(* Logix 5000 project; controller Comas_L4 vendor 1 type 14 code 193 rev 30.11; software revision 30.02 *)

TASK Gestion_Rapide (task) : Main
TASK MainTask (periodic, rate 5 ms, priority 10, watchdog 10 ms) : General, Comas

MODULES
   Local : vendor 1 type 14 code 193 (5069 0, rev 30.11)
      SortieF_4 : vendor 1 type 14 code 154 (Ethernet 172.10.3.20, rev 21.1)
      Var_Vertical_Droit : vendor 1 type 37 code 48 (Ethernet 172.10.12.22, rev 7.1, MotionDiagnostics RPI 1 ms, MotionSync RPI 5 ms)
      Var_Pompe_Doseuse : vendor 1 type 37 code 49 (Ethernet 172.10.12.20, rev 7.1, MotionSync RPI 5 ms, MotionDiagnostics RPI 1 ms)
      Var_Vertical_Gauche : vendor 1 type 37 code 48 (Ethernet 172.10.12.21, rev 7.1, MotionSync RPI 5 ms, MotionDiagnostics RPI 1 ms)
      Var_Rouleaux_Canneles : vendor 1 type 37 code 48 (Ethernet 172.10.12.26, rev 7.1, MotionDiagnostics RPI 1 ms, MotionSync RPI 5 ms)
      Codeur_Four : 842E-CM-M (Ethernet 172.10.12.19, rev 1.1, MotionDiagnostics RPI 1 ms, MotionSync RPI 5 ms)
      Var_Coupe_Fil : vendor 1 type 37 code 48 (Ethernet 172.10.12.25, rev 7.1, MotionSync RPI 5 ms, MotionDiagnostics RPI 1 ms)
      Var_Horizontal_Gauche : vendor 1 type 37 code 48 (Ethernet 172.10.12.23, rev 7.1, MotionSync RPI 5 ms, MotionDiagnostics RPI 1 ms)
      Var_Horizontal_Droit : vendor 1 type 37 code 48 (Ethernet 172.10.12.24, rev 7.1, MotionDiagnostics RPI 1 ms, MotionSync RPI 5 ms)
      Stratix_5700 : vendor 1 type 12 code 241 (Ethernet 172.10.12.13, rev 7.1, Output RPI 1000 ms)
      Entrees_2 : 5069-IB16 (5069 2, rev 2.1, StandardDataDriven RPI 5 ms)
      Entrees_1 : 5069-IB16 (5069 1, rev 2.1, StandardDataDriven RPI 5 ms)
      Sorties_1 : 5069-OB16 (5069 3, rev 2.1, StandardDataDriven RPI 5 ms)
END_MODULES

TYPE Chart :   // Chart Control Data Source
STRUCT
   Title : STRING;
   NumberOfDataPoints : INT;
   X_Axis_Label : STRING;
   X_Axis_Min : REAL;
   X_Axis_Max : REAL;
   Y_Axis_Label : STRING;
   Y_Axis_Min : REAL;
   Y_Axis_Max : REAL;
   DataSeries_FixedAxis : DataSeries;
   DataSeries_1 : DataSeries;
   DataSeries_2 : DataSeries;
   DataSeries_3 : DataSeries;
   DataSeries_4 : DataSeries;
   DataSeries_5 : DataSeries;
   DataSeries_6 : DataSeries;
   DataSeries_7 : DataSeries;
   DataSeries_8 : DataSeries;
END_STRUCT
END_TYPE

TYPE DataSeries :
STRUCT
   Label : STRING;
   Visible : BOOL;
   Data : REAL[500];
END_STRUCT
END_TYPE

TYPE UDT_Axis_Cam_Profil :
STRUCT
   Cam : CAM[80];
   MasterPeriode : REAL;
   SlavePeriode : REAL;
   NbrOfCamPoints : DINT;
   StartSlope : REAL;
   EndSlope : REAL;
   MasterScaling : REAL;
   SlaveScaling : REAL;
END_STRUCT
END_TYPE

TYPE UDT_CAM_PAN :
STRUCT
   A : UDT_CAM_POINT;
   B : UDT_CAM_POINT;
   C : UDT_CAM_POINT;
   D : UDT_CAM_POINT;
   E : UDT_CAM_POINT;
   F : UDT_CAM_POINT;
   G : UDT_CAM_POINT;
   H : UDT_CAM_POINT;
   I : UDT_CAM_POINT;
   J : UDT_CAM_POINT;
   K : UDT_CAM_POINT;
   L : UDT_CAM_POINT;
   M : UDT_CAM_POINT;
   N : UDT_CAM_POINT;
   O : UDT_CAM_POINT;
   P : UDT_CAM_POINT;
   Q : UDT_CAM_POINT;
   R : UDT_CAM_POINT;
   S : UDT_CAM_POINT;
   T : UDT_CAM_POINT;
   U : UDT_CAM_POINT;
   V : UDT_CAM_POINT;
   W : UDT_CAM_POINT;
   X : UDT_CAM_POINT;
   Y : UDT_CAM_POINT;
END_STRUCT
END_TYPE

TYPE UDT_CAM_POINT :
STRUCT
   x : REAL;
   y : REAL;
END_STRUCT
END_TYPE

TYPE UDT_CamGeneration :
STRUCT
   Cmd : UDT_CamGeneration_Cmd;
   In : UDT_CamGeneration_In;
   Out : UDT_CamGeneration_Out;
END_STRUCT
END_TYPE

TYPE UDT_CamGeneration_Cmd :
STRUCT
   Reset : BOOL;   // Effacement défaut
   Start : BOOL;   // Commande de lancement des calculs
   CamOrCamProfil : BOOL;   // 0 = tableau de points (sans MCCP) 1 = Profil executable (avec MCCP)
   Optimize : BOOL;
END_STRUCT
END_TYPE

TYPE UDT_CamGeneration_In :
STRUCT
   Cam : CAM[32];
   StartSlope : REAL;
   EndSlope : REAL;
   DefaultProfilType : INT;   // 2 = Modified Trapezoidal 4 = Sine modified 5 = 3-4-5 Poly 7 = 4-5-6-7 Poly
   Cfg_Segments : UDT_SegmentSetUp[32];
END_STRUCT
END_TYPE

TYPE UDT_CamGeneration_Out :
STRUCT
   Cam : CAM[32];
   NbrOfCamPoints : DINT;
   StartSlope : REAL;
   EndSlope : REAL;
   CamProfil : CAM_PROFILE[32];
END_STRUCT
END_TYPE

TYPE UDT_CamSegment :
STRUCT
   M0 : REAL;
   S0 : REAL;
   V0 : REAL;
   V1 : REAL;
   V2 : REAL;
   M1 : REAL;
   M2 : REAL;
   M3 : REAL;
   M4 : REAL;
   M5 : REAL;
   dM : REAL;
   a4 : REAL;
   S1 : REAL;
   S2 : REAL;
   S3 : REAL;
   S4 : REAL;
   S5 : REAL;
   dS : REAL;
   K1 : REAL;
   K2 : REAL;
   K3 : REAL;
   K4 : REAL;
   K5 : REAL;
   K6 : REAL;
   K7 : REAL;
   K8 : REAL;
   K9 : REAL;
   ActSlope : REAL;
   PrevSlope : REAL;
   No_Of_Points : DINT;
   NbPoints : DINT;
   CfgIndex : DINT;
   CAM_Points : CAM[32];
   Cv : REAL[2];
   Mn : REAL[2];
   Sn : REAL[2];
   RiseReturnComp : BOOL[32];
   IsAcceleration : BOOL;
   Err : BOOL;
   B1 : BOOL;
   MemoRiseReturnComp : BOOL;
END_STRUCT
END_TYPE

TYPE UDT_COM_Comas_Vers_SortieF :   // echange de donnée entre comas et sortie four
STRUCT
   Forage_Panel_O_F_Trappe : BOOL;
   ReserveBool : BOOL;
   ReserveBool2 : BOOL;
   ReserveReal : REAL;
   ReserveReal2 : REAL;
   ReserveReal3 : REAL;
END_STRUCT
END_TYPE

TYPE UDT_COMAS :
STRUCT
   Pas_Machine : DINT;
   Dephasage_Maitre : REAL;
   Came_Maitre : CAM[100];
   Longueur_Came_Maitre : DINT;
   Tete : UDT_COMAS_TETE;
   Pompe : UDT_COMAS_POMPE;
   Rouleaux : UDT_COMAS_ROULEAUX;
   Coupe_Fil : UDT_COMAS_COUPE;
   Start_Cam_Logique_Decoreuse : REAL;
   Stop_Cam_Logique_Decoreuse : REAL;
   Start_Cam_Logique_Doseuse : REAL;
   Stop_Cam_Logique_Doseuse : REAL;
   Consigne_Vitesse_Manu_mm : REAL;
   Consigne_Acc_Decc_Manu_mm : REAL;
   Consigne_Jerk_Manu : REAL;
   Activation_Cam_Auto : BOOL;
   Mode_CPT_Presence : BOOL;
   Distance_CPT_Presence_Produit : DINT;
   Consigne_Vitesse_Manu_Tour : REAL;
   Consigne_Acc_Decc_Manu_Tour : REAL;
   Distance_Decoreuse_mm : REAL;
   Distance_Doseuse_mm : REAL;
   Mode_Decoreuse_Cam_Logique : BOOL;
   Reserve_Real1 : REAL;
   Reserve_Real2 : REAL;
   Reserve_Real3 : REAL;
   Reserve_Real4 : REAL;
   Reserve_Real5 : REAL;
   Reserve_Bool1 : BOOL;
   Reserve_Bool2 : BOOL;
   Reserve_Bool3 : BOOL;
   Reserve_Bool4 : BOOL;
   Reserve_Bool5 : BOOL;
   Reserve_Real6 : REAL;
   Reserve_Real7 : REAL;
   Reserve_Real8 : REAL;
   Reserve_Real9 : REAL;
   Reserve_Real10 : REAL;
END_STRUCT
END_TYPE

TYPE UDT_COMAS_COUPE :
STRUCT
   Activation : BOOL;
   Start_Cam_Logique_Virtuelle : REAL;
   Stop_Cam_Logique_Virtuelle : REAL;
   Consigne_Vitesse_Virtuelle : REAL;
   Consigne_Acc_Dec_Virtuelle : REAL;
   Consigne_Jerk_Virtuelle : REAL;
   Cam_Axe : CAM[100];
   Longueur_Cam_Axe : DINT;
   Offset_Axe : REAL;
   Points_Pan : UDT_CAM_PAN;
   Reserve_Real1 : REAL;
   Reserve_Real2 : REAL;
   Reserve_Real3 : REAL;
   Reserve_Real4 : REAL;
   Reserve_Real5 : REAL;
   Reserve_Bool1 : BOOL;
   Reserve_Bool2 : BOOL;
   Reserve_Bool3 : BOOL;
   Reserve_Bool4 : BOOL;
   Reserve_Bool5 : BOOL;
END_STRUCT
END_TYPE

TYPE UDT_COMAS_POMPE :
STRUCT
   Start_Cam_Logique_Avance : REAL;
   Stop_Cam_Logique_Avance : REAL;
   Start_Cam_Logique_Recul : REAL;
   Stop_Cam_Logique_Recul : REAL;
   Consigne_Vitesse_Avance : REAL;
   Consigne_Acc_Dec_Avance : REAL;
   Consigne_Jerk_Avance : REAL;
   Consigne_Vitesse_Recul : REAL;
   Consigne_Acc_Dec_Recul : REAL;
   Consigne_Jerk_Recul : REAL;
   Offset_Axe : REAL;
   Points_Pan : UDT_CAM_PAN;
   Start_Cam_Logique_Inter1 : REAL;
   Stop_Cam_Logique_Inter1 : REAL;
   Consigne_Vitesse_Inter1 : REAL;
   Start_Cam_Logique_Inter2 : REAL;
   Stop_Cam_Logique_Inter2 : REAL;
   Consigne_Vitesse_Inter2 : REAL;
   Start_Cam_Logique_Inter3 : REAL;
   Stop_Cam_Logique_Inter3 : REAL;
   Consigne_Vitesse_Inter3 : REAL;
   Start_Cam_Logique_Inter4 : REAL;
   Stop_Cam_Logique_Inter4 : REAL;
   Consigne_Vitesse_Inter4 : REAL;
   Start_Cam_Logique_Inter5 : REAL;
   Stop_Cam_Logique_Inter5 : REAL;
   Consigne_Vitesse_Inter5 : REAL;
   Start_Cam_Logique_Inter6 : REAL;
   Stop_Cam_Logique_Inter6 : REAL;
   Consigne_Vitesse_Inter6 : REAL;
   Start_Cam_Logique_Inter7 : REAL;
   Stop_Cam_Logique_Inter7 : REAL;
   Consigne_Vitesse_Inter7 : REAL;
   Start_Cam_Logique_Inter8 : REAL;
   Stop_Cam_Logique_Inter8 : REAL;
   Consigne_Vitesse_Inter8 : REAL;
   Reserve_Real1 : REAL;
   Reserve_Real2 : REAL;
   Reserve_Real3 : REAL;
   Reserve_Real4 : REAL;
   Reserve_Real5 : REAL;
   Reserve_Bool1 : BOOL;
   Reserve_Bool2 : BOOL;
   Reserve_Bool3 : BOOL;
   Reserve_Bool4 : BOOL;
   Reserve_Bool5 : BOOL;
END_STRUCT
END_TYPE

TYPE UDT_COMAS_ROULEAUX :
STRUCT
   Syncho_Pompe : BOOL;
   Consigne_Vitesse : REAL;
   Consigne_Acc_Dec : REAL;
   Consigne_Jerk : REAL;
   Offset_Axe : REAL;
   Reserve_Real1 : REAL;
   Reserve_Real2 : REAL;
   Reserve_Real3 : REAL;
   Reserve_Real4 : REAL;
   Reserve_Real5 : REAL;
   Reserve_Bool1 : BOOL;
   Reserve_Bool2 : BOOL;
   Reserve_Bool3 : BOOL;
   Reserve_Bool4 : BOOL;
   Reserve_Bool5 : BOOL;
END_STRUCT
END_TYPE

TYPE UDT_COMAS_TETE :
STRUCT
   Start_Cam_Logique_Degagement : REAL;
   Stop_Cam_Logique_Degagement : REAL;
   Position_Degagement_H : REAL;
   Position_Degagement_V : REAL;
   Centrage_Tete : INT;
   Hauteur_Tete : INT;
   Cam_Axe_Horizontal : CAM[100];
   Cam_Axe_Vertical : CAM[100];
   Longueur_Cam_Axe_H : DINT;
   Longueur_Cam_Axe_V : DINT;
   Offset_Vertical_Gauche : REAL;
   Offset_Horizontal_Gauche : REAL;
   Cam_Axe_Horizontal_Pan : UDT_CAM_PAN;
   Cam_Axe_Vertical_Pan : UDT_CAM_PAN;
   Offset_Vertical_Droit : REAL;
   Offset_Horizontal_Droit : REAL;
   Reserve_Real1 : REAL;
   Reserve_Real2 : REAL;
   Reserve_Real3 : REAL;
   Reserve_Real4 : REAL;
   Reserve_Real5 : REAL;
   Reserve_Bool1 : BOOL;
   Reserve_Bool2 : BOOL;
   Reserve_Bool3 : BOOL;
   Reserve_Bool4 : BOOL;
   Reserve_Bool5 : BOOL;
END_STRUCT
END_TYPE

TYPE UDT_HMI :
STRUCT
   Index_Recette_a_sauver : DINT;
   Index_Recette_a_charger : DINT;
   Index_Recette_en_cours : DINT;
   Index_Recette_a_supprimer : DINT;
   BP_Valid_Recette : BOOL;
   BP_Sauve_Recette : BOOL;
   BP_Sup_Recette : BOOL;
END_STRUCT
END_TYPE

TYPE UDT_RECIPE :
STRUCT
   Name : STRING;
   Comas : UDT_COMAS;
   Reserve_Real1 : REAL;
   Reserve_Real2 : REAL;
   Reserve_Real3 : REAL;
   Reserve_Real4 : REAL;
   Reserve_Real5 : REAL;
   Reserve_Bool1 : BOOL;
   Reserve_Bool2 : BOOL;
   Reserve_Bool3 : BOOL;
   Reserve_Bool4 : BOOL;
   Reserve_Bool5 : BOOL;
END_STRUCT
END_TYPE

TYPE UDT_REGISTRE_TAPIS :
STRUCT
   Position : REAL;
   Etat_Produit : DINT;   // bit 0 -> 1=produit traité par l'API et 0=non traité
   Reserve_Real1 : REAL;
   Reserve_Real2 : REAL;
   Reserve_Real3 : REAL;
   Reserve_Real4 : REAL;
   Reserve_Real5 : REAL;
   Reserve_Bool1 : BOOL;
   Reserve_Bool2 : BOOL;
   Reserve_Bool3 : BOOL;
   Reserve_Bool4 : BOOL;
   Reserve_Bool5 : BOOL;
END_STRUCT
END_TYPE

TYPE UDT_SegmentSetUp :
STRUCT
   AccelProportion : REAL;   // X means 1/X accel
   DecelProportion : REAL;   // X means 1/X decel
   ProfilType : INT;   // 2 = Modified Trapezoidal 4 = Sine modified 5 = 3-4-5 Poly 7 = 4-5-6-7 Poly
END_STRUCT
END_TYPE

ADD_ON_INSTRUCTION AOI_CamDisplay_OCX_StdCAM   (* revision 1.2, ExecutePrescan, ExecuteEnableInFalse *)
// Revision note:
// 1.1 :
// - Review Scaling for velocity and acceleration chart
// 1.2 :
// - Correct the checksum calculation
VAR_IN_OUT
   MIO_CAM : UDT_Axis_Cam_Profil; {required}
   MIO_CAMDisplay : Chart; {required}
END_VAR
VAR_OUTPUT
   Sts_EN : BOOL; {access Read Only, visible}
   Sts_ER : BOOL; {access Read Only, visible}
   Sts_ERR : DINT; {access Read Only, visible}
   Sts_EXERR : DINT; {access Read Only, visible}
END_VAR
VAR_INPUT
   In_ClearFault : BOOL; {visible}
END_VAR
VAR
   L_Sequence : DINT;
   L_CAMIndex : DINT; {access None}
   L_MI_MCCP : MOTION_INSTRUCTION; {access None}
   L_CAMProfile : CAM_PROFILE[80]; {access None}
   L_MI_MCSV : MOTION_INSTRUCTION; {access None}
   L_Inc : REAL; {access None}
   L_Master : REAL; {access None}
   L_OldNbPoints : DINT; {access None}
   L_OldProfDisplay : DINT; {access None}
   L_MaxPos : REAL; {access Read Only}
   L_MinPos : REAL; {access Read Only}
   L_MaxVel : REAL; {access Read Only}
   L_MinVel : REAL; {access Read Only}
   L_MaxAcc : REAL; {access Read Only}
   L_MinAcc : REAL; {access Read Only}
   L_StartVal : DINT; {access None}
   L_EndVal : DINT; {access None}
   L_ScaleVel : REAL; {access None}
   L_ScaleAcc : REAL; {access None}
   Min1 : REAL; {access None}
   Min2 : REAL; {access None}
   L_OldCheckSum : REAL; {access None}
   L_I : DINT; {access None}
   L_CheckSum : REAL; {access None}
   Max1 : REAL; {access None}
   Max2 : REAL; {access None}
   L_Array_Size : DINT; {access None}
   L_Cam_Visu : CAM[80]; {access None}
END_VAR

ROUTINE EnableInFalse   (* structured text *)
   L_Sequence 					:= 0;
   Sts_EN 						:= 0;
   Sts_ER 						:= 0;
   L_Master					:= 0;
   L_MI_MCSV.FLAGS				:= 0;
   L_OldNbPoints				:= 0;
   L_OldProfDisplay			:= -1;
   
END_ROUTINE

ROUTINE Logic   (* structured text *)
   
   Case L_Sequence of
   
   00: If (MIO_CAM.NbrOfCamPoints > 0) Then
   		L_CheckSum := 0 ;
   		For L_I := 0 To (MIO_CAM.NbrOfCamPoints-1) Do
   			L_CheckSum						:= MIO_CAM.Cam[L_I].Master
   											+ MIO_CAM.Cam[L_I].Slave
   											+ MIO_CAM.Cam[L_I].SegmentType
   											+ L_CheckSum;
   		End_For;
   		L_CheckSum := L_CheckSum + MIO_CAM.SlaveScaling + MIO_CAM.MasterScaling;
   		If (L_CheckSum <> L_OldCheckSum) Then
   			Sts_ER 								:= 0;
   			L_MI_MCCP.FLAGS						:= 0;
   			L_OldCheckSum						:= L_CheckSum;
   			L_OldNbPoints						:= MIO_CAM.NbrOfCamPoints;
   			L_MaxPos							:= -1000;
   			L_MinPos							:= 1000;
   			L_MaxVel							:= -1000;
   			L_MinVel							:= 1000;
   			L_MaxAcc							:= -1000;
   			L_MinAcc							:= 1000;
   			L_OldProfDisplay					:= 0;
   			MIO_CAMDisplay.NumberOfDataPoints	:= 130;
   			L_Sequence							:= 5;
   		End_If;
   	End_If;
   
   5:	For L_I := 0 To L_Array_Size-1 Do
   			L_Cam_Visu[L_I].Slave			:= MIO_CAM.Cam[L_I].Slave *  MIO_CAM.SlaveScaling;
   			L_Cam_Visu[L_I].Master			:= MIO_CAM.Cam[L_I].Master * MIO_CAM.MasterScaling;
   			L_Cam_Visu[L_I].SegmentType		:= MIO_CAM.Cam[L_I].SegmentType;
   	End_For;
   	L_Sequence								:= 10;
   
   
   10: MCCP(L_MI_MCCP,L_Cam_Visu[0],L_OldNbPoints,MIO_CAM.StartSlope,MIO_CAM.EndSlope,L_CAMProfile);
   	If L_MI_MCCP.DN Then
   		MIO_CAMDisplay.X_Axis_Min			:= L_Cam_Visu[0].Master;
   		MIO_CAMDisplay.X_Axis_Max			:= L_Cam_Visu[L_OldNbPoints-1].Master;
   		L_Master							:= MIO_CAMDisplay.X_Axis_Min;
   		L_Inc								:= (MIO_CAMDisplay.X_Axis_Max - MIO_CAMDisplay.X_Axis_Min) / 130;
   		L_StartVal							:= 0;
   		L_EndVal							:= 25;
   		L_Sequence 							:= 20;
   	Elsif L_MI_MCCP.ER Then
   		Sts_ER 								:= 1;
   		Sts_ERR 							:= L_MI_MCCP.ERR;
   		Sts_EXERR 							:= L_MI_MCCP.EXERR;
   		L_Sequence 							:= 99;
   	End_if;
   
   20:	For L_CAMIndex := L_StartVal to L_EndVal Do
   		L_MI_MCSV.FLAGS						:= 0;
   		MCSV(L_MI_MCSV,L_CAMProfile,L_Master,MIO_CAMDisplay.DataSeries_1.Data[L_CAMIndex],MIO_CAMDisplay.DataSeries_2.Data[L_CAMIndex],MIO_CAMDisplay.DataSeries_3.Data[L_CAMIndex]);
   		MIO_CAMDisplay.DataSeries_FixedAxis.Data[L_CAMIndex] := L_Master;
   		If 	L_MI_MCSV.ER Then
   			Sts_ER 							:= 1;
   			Sts_ERR 						:= L_MI_MCSV.ERR;
   			Sts_EXERR						:= L_MI_MCSV.EXERR;
   			Exit;
   			L_Sequence 						:= 99;
   		Else
   			If L_CAMIndex < 128 Then
   				L_Master					:= L_Master + L_Inc;
   			Else
   				L_Master					:= MIO_CAMDisplay.X_Axis_Max;
   			End_If;
   			If MIO_CAMDisplay.DataSeries_1.Data[L_CAMIndex] > L_MaxPos Then
   				L_MaxPos					:= MIO_CAMDisplay.DataSeries_1.Data[L_CAMIndex];
   			End_If;
   			If MIO_CAMDisplay.DataSeries_1.Data[L_CAMIndex] < L_MinPos Then
   				L_MinPos					:= MIO_CAMDisplay.DataSeries_1.Data[L_CAMIndex];
   			End_If;
   			If MIO_CAMDisplay.DataSeries_2.Data[L_CAMIndex] > L_MaxVel Then
   				L_MaxVel					:= MIO_CAMDisplay.DataSeries_2.Data[L_CAMIndex];
   			End_If;
   			If MIO_CAMDisplay.DataSeries_2.Data[L_CAMIndex] < L_MinVel Then
   				L_MinVel					:= MIO_CAMDisplay.DataSeries_2.Data[L_CAMIndex];
   			End_If;
   			If MIO_CAMDisplay.DataSeries_3.Data[L_CAMIndex] > L_MaxAcc Then
   				L_MaxAcc					:= MIO_CAMDisplay.DataSeries_3.Data[L_CAMIndex];
   			End_If;
   			If MIO_CAMDisplay.DataSeries_3.Data[L_CAMIndex] < L_MinAcc Then
   				L_MinAcc					:= MIO_CAMDisplay.DataSeries_3.Data[L_CAMIndex];
   			End_If;
   		End_If;
   	End_For;
   	If Not L_MI_MCSV.ER Then
   		If L_CAMIndex >= 129 Then
   			L_Sequence						:= 30;
   		Else
   			L_Sequence						:= 25;
   		End_If;
   	End_If;
   
   25: L_StartVal								:= L_EndVal + 1;
   	L_EndVal								:= L_EndVal + 26;
   	L_Sequence								:= 20;
   
   30: If (L_MaxVel = 0) And (L_MinVel = L_MaxVel) Then
   		L_ScaleVel							:= 0;
   		L_ScaleAcc							:= 0;
   	Elsif (L_MaxVel <> 0) And (L_MinVel = L_MaxVel) Then
   		L_ScaleVel							:= ((L_MaxPos - L_MinPos) / 2)/L_MaxVel;
   		L_ScaleAcc							:= 0;
   	Else
   		L_ScaleVel							:= (L_MaxPos - L_MinPos) / (L_MaxVel - L_MinVel);
   		L_ScaleAcc							:= (L_MaxPos - L_MinPos) / (L_MaxAcc - L_MinAcc);
   	End_If;
   	L_StartVal								:= 0;
   	L_EndVal								:= 25;
   	L_Sequence 								:= 31;
   
   31: For L_CAMIndex := L_StartVal to L_EndVal Do
   		MIO_CAMDisplay.DataSeries_2.Data[L_CAMIndex]	:= MIO_CAMDisplay.DataSeries_2.Data[L_CAMIndex] * L_ScaleVel;
   		MIO_CAMDisplay.DataSeries_3.Data[L_CAMIndex]	:= MIO_CAMDisplay.DataSeries_3.Data[L_CAMIndex] * L_ScaleAcc;
   	End_For;
   	If L_CAMIndex >= 129 Then
   		L_Sequence							:= 40;
   	Else
   		L_Sequence							:= 32;
   	End_If;
   
   32:	L_StartVal								:= L_EndVal + 1;
   	L_EndVal								:= L_EndVal + 26;
   	L_Sequence								:= 31;
   
   40: Min1	:= L_MinVel*L_ScaleVel;
   	Min2	:= L_MinAcc*L_ScaleAcc;
   	//Calculate Minimum value to display
   	//If velocity value is the minimum
   	If Min1 < Min2 AND Min1 <= L_MinPos Then
   		MIO_CAMDisplay.Y_Axis_Min			:= Min1;
   	//If acceleration value is the minimum
   	Elsif Min2 < Min1 AND Min2 <= L_MinPos Then
   		MIO_CAMDisplay.Y_Axis_Min			:= Min2;
   	//If position value is the minimum
   	Elsif L_MinPos < Min1 AND L_MinPos < Min2 Then
   		MIO_CAMDisplay.Y_Axis_Min			:= L_MinPos;
   	Elsif Min1 = Min2 Then
   		MIO_CAMDisplay.Y_Axis_Min			:= -0.1;
   	End_If;
   
   	Max1	:= L_MaxVel*L_ScaleVel;
   	Max2	:= L_MaxAcc*L_ScaleAcc;
   	//Calculate Maximum value to display
   	//If velocity value is the maximum
   	If Max1 > Max2 AND Max1 >= L_MaxPos Then
   		MIO_CAMDisplay.Y_Axis_Max			:= Max1;
   	//If acceleration value is the maximum
   	Elsif Max2 > Max1 AND Max2 >= L_MaxPos Then
   		MIO_CAMDisplay.Y_Axis_Max			:= Max2;
   	//If position value is the maximum
   	Elsif L_MaxPos > Max1 AND L_MaxPos > Max2 Then
   		MIO_CAMDisplay.Y_Axis_Max			:= L_MaxPos;
   	Elsif Max1 = Max2 Then
   		MIO_CAMDisplay.Y_Axis_Max			:= 0.1;
   	End_If;
   
   
   	MIO_CAMDisplay.DataSeries_1.Visible		:= 1;
   	MIO_CAMDisplay.DataSeries_2.Visible		:= 1;
   	MIO_CAMDisplay.DataSeries_3.Visible		:= 1;
   
   	L_Sequence								:= 0;
   
   99: If In_ClearFault Then
   		Sts_ER 								:= 0;
   		L_MI_MCCP.FLAGS						:= 0;
   		L_MI_MCSV.FLAGS						:= 0;
   		Sts_ERR 							:= 0;
   		Sts_EXERR							:= 0;
   		L_Sequence							:= 0;
   	End_If;
   End_Case;
   
   Sts_EN	:= EnableIn;
END_ROUTINE

ROUTINE Prescan   (* structured text *)
   L_Sequence 					:= 0;
   Sts_EN 						:= 0;
   Sts_ER 						:= 0;
   L_Master					:= 0;
   L_MI_MCSV.FLAGS				:= 0;
   L_OldNbPoints				:= 0;
   L_OldProfDisplay			:= -1;
   MIO_CAMDisplay.DataSeries_FixedAxis.Visible :=1;
   MIO_CAMDisplay.DataSeries_1.Label := 'Position';
   MIO_CAMDisplay.DataSeries_2.Label := 'Velocity';
   MIO_CAMDisplay.DataSeries_3.Label := 'Acceleration';
   Size(L_CAMProfile,0,L_Array_Size);
END_ROUTINE
END_ADD_ON_INSTRUCTION

ADD_ON_INSTRUCTION AOI_CamGenerator_ST   (* revision 24.0, ExecutePrescan *)
VAR_IN_OUT
   MIO_CAM_Interface : UDT_CamGeneration; {required}
END_VAR
VAR_OUTPUT
   Sts_ERR : DINT; {access Read Only, visible}
   Sts_EXERR : DINT; {access Read Only, visible}
   Sts_IP : BOOL; {access Read Only, visible}
   Sts_PC : BOOL; {access Read Only, visible}
   Sts_ER : BOOL; {access Read Only, visible}
   CycleTime : DINT; {access Read Only}
   L_NbCAMPoints : DINT; {access Read Only}
END_VAR
VAR
   CAM_Design : UDT_CamSegment;
   L_CAMIndex : DINT; {access None}
   L_I : DINT; {access None}
   L_AOI_CAM_PosComp : AOI_PosComp_ST; {access None}
   L_MI_MCCP : MOTION_INSTRUCTION; {access None}
   L_SlvVal : REAL; {access None}
   L_SlvAcc : REAL; {access None}
   L_MI_MCSV : MOTION_INSTRUCTION; {access None}
   L_InLength : DINT; {access None}
   L_NbSegToTransf : DINT; {access None}
   L_V2 : REAL[800]; {access None}
   L_OutLength : DINT; {access None}
   L_CheckSum : REAL; {access None}
   L_OldCheckSum : REAL; {access None}
   CST : DINT[4]; {access None}
   L_FirstSlope : BOOL; {access None}
   L_SndSlope : BOOL; {access None}
   L_Optimize : BOOL; {access None}
   L_Rebuilt : BOOL; {access None}
   L_Slope1 : REAL; {access None}
   L_Slope2 : REAL; {access None}
   L_DSlope : REAL; {access None}
   L_CAMLength : DINT; {access None}
   L_CAMPLength : DINT; {access None}
END_VAR

ROUTINE Logic   (* structured text *)
   // Clear fault
   If MIO_CAM_Interface.Cmd.Reset And Sts_ER Then
   	Sts_ER 					:= 0;
   	Sts_ERR					:= 0;
   	Sts_EXERR 				:= 0;
   	CAM_Design.Err			:= 0;
   End_If;
   //Wait for start
   If Not MIO_CAM_Interface.Cmd.Start Then
   	Sts_PC 					:= 0;
   	TND();
   Elsif Sts_ER Or (MIO_CAM_Interface.Cmd.Start And Sts_PC) Then
   	TND();
   End_If;
   
   GSV(CST,,CurrentValue,CST[0]);
   
   //--------------------------------------------------
   //				Cam Generation execution
   //--------------------------------------------------
   Sts_IP 						:= 1;
   CAM_Design.No_Of_Points 	:= 0;
   L_MI_MCCP.FLAGS 			:= 0;
   L_NbSegToTransf				:= 0;
   L_NbCAMPoints 				:= 1;
   L_CheckSum					:= 0;
   
   IF Not MIO_CAM_Interface.Cmd.CamOrCamProfil Then
   	L_OutLength := L_CAMLength;
   Else
   	L_OutLength := L_CAMPLength;
   End_If;
   
   For L_I:= 0 to (L_OutLength - 1) Do
   	MIO_CAM_Interface.Out.Cam[L_I].Master 					:= 0;
   	MIO_CAM_Interface.Out.Cam[L_I].Slave 					:= 0;
   	MIO_CAM_Interface.Out.Cam[L_I].SegmentType 				:= 0;
   End_For;
   
   // Check Cam Length
   For L_I:= 1 to (L_InLength - 1) Do
   	L_CheckSum			:= MIO_CAM_Interface.In.Cam[L_I-1].Master + MIO_CAM_Interface.In.Cam[L_I-1].Slave + MIO_CAM_Interface.In.Cam[L_I-1].SegmentType + L_CheckSum;
   	If MIO_CAM_Interface.In.DefaultProfilType <> -1 Then
   		MIO_CAM_Interface.In.Cfg_Segments[L_I-1].ProfilType	:= MIO_CAM_Interface.In.DefaultProfilType;
   	End_If;
   	If MIO_CAM_Interface.In.Cam[L_I].Master <> 0 Then
   		L_NbCAMPoints	:= L_NbCAMPoints + 1;
   	Else
   		Exit;
   	End_If;
   End_For;
   
   If (MIO_CAM_Interface.Cmd.Optimize And Not L_Optimize) Then
   	L_Rebuilt	:= 1;
   	L_Optimize	:= 1;
   Elsif (Not MIO_CAM_Interface.Cmd.Optimize And L_Optimize) Then
   	L_Rebuilt	:= 1;
   	L_Optimize	:= 0;
   End_If;
   
   // Compute PCAM
   If (L_CheckSum <> L_OldCheckSum) Or L_Rebuilt Then
   	MCCP(L_MI_MCCP,
   		MIO_CAM_Interface.In.Cam,
   		L_NbCAMPoints,
   		MIO_CAM_Interface.In.StartSlope,
   		MIO_CAM_Interface.In.EndSlope,
   		MIO_CAM_Interface.Out.CamProfil);
   
   	If L_MI_MCCP.ER Then
   		Sts_IP 					:= 0;
   		Sts_ER 					:= 1;
   		Sts_ERR 				:= L_MI_MCCP.ERR;
   		Sts_EXERR 				:= L_MI_MCCP.EXERR;
   		TND();
   	End_if;
   
   	//Examine number of Cam points needed
   	For L_I:= 1 to (L_NbCAMPoints-1) Do
   		L_MI_MCSV.FLAGS			:= 0;
   		MCSV(L_MI_MCSV,
   			MIO_CAM_Interface.Out.CamProfil,
   			MIO_CAM_Interface.In.Cam[L_I].Master,
   			L_SlvVal,
   			L_V2[L_I],
   			L_SlvAcc);
   		If (MIO_CAM_Interface.In.Cam[L_I-1].SegmentType = 1) And (MIO_CAM_Interface.In.Cfg_Segments[L_I-1].ProfilType <> 0) Then
   			L_NbSegToTransf								:= L_NbSegToTransf + 1;
   			If (L_I < (L_NbCAMPoints-1)) And MIO_CAM_Interface.Cmd.Optimize Then
   				L_FirstSlope	:= (MIO_CAM_Interface.In.Cam[L_I].Slave >= MIO_CAM_Interface.In.Cam[L_I-1].Slave);
   				L_SndSlope		:= (MIO_CAM_Interface.In.Cam[L_I+1].Slave >= MIO_CAM_Interface.In.Cam[L_I].Slave);
   				If ((L_FirstSlope And Not L_SndSlope) Or (Not L_FirstSlope And L_SndSlope)) And (L_V2[L_I] <> 0) Then
   					L_V2[L_I] := 0;
   				Else
   					L_Slope1	:= (MIO_CAM_Interface.In.Cam[L_I].Slave - MIO_CAM_Interface.In.Cam[L_I-1].Slave) / (MIO_CAM_Interface.In.Cam[L_I].Master - MIO_CAM_Interface.In.Cam[L_I-1].Master);
   					L_Slope2	:= (MIO_CAM_Interface.In.Cam[L_I+1].Slave - MIO_CAM_Interface.In.Cam[L_I].Slave) / (MIO_CAM_Interface.In.Cam[L_I+1].Master - MIO_CAM_Interface.In.Cam[L_I].Master);
   					If (L_Slope1 <> 0) And (L_Slope2 <> 0) Then
   						L_DSlope							:= L_Slope1 / L_Slope2;
   					Else
   						L_DSlope							:= 0;
   					End_If;
   					If ABS(L_DSlope) > 3 Then
   						L_V2[L_I] := L_V2[L_I] /(L_DSlope/2.8);
   					End_If;
   				End_If;
   				CAM_Design.RiseReturnComp[L_I-1]		:= ((L_FirstSlope And Not L_SndSlope) Or (Not L_FirstSlope And L_SndSlope) Or (MIO_CAM_Interface.In.Cam[L_I-1].SegmentType = MIO_CAM_Interface.In.Cam[L_I].SegmentType)) And ((MIO_CAM_Interface.In.Cam[L_I].SegmentType = 1) And (MIO_CAM_Interface.In.Cfg_Segments[L_I-1].ProfilType <> 3));
   			Else
   				CAM_Design.RiseReturnComp[L_I-1]		:= 0;
   			End_If;
   		Else
   			L_FirstSlope								:= 0;
   			L_SndSlope									:= 0;
   			CAM_Design.RiseReturnComp[L_I-1]			:= 0;
   		End_If;
   	End_For;
   
   	If L_NbSegToTransf > 0 Then
   		CAM_Design.NbPoints		:= ((L_OutLength - (L_NbCAMPoints - L_NbSegToTransf))/L_NbSegToTransf) - 2;
   	Else
   		CAM_Design.NbPoints 	:= 15;
   	End_If;
   
   	If (CAM_Design.NbPoints > 15) Then
   		CAM_Design.NbPoints 	:= 15;
   	Elsif (CAM_Design.NbPoints < 5) Then
   		Sts_ERR					:= 190;
   		Sts_EXERR				:= 0;
   		Sts_ER					:= 1;
   		Sts_IP					:= 0;
   		TND();
   	End_If;
   	L_OldCheckSum				:= L_CheckSum;
   	L_Rebuilt					:= 0;
   End_If;
   
   //Generate PCAM
   For L_CAMIndex := 1 to (L_NbCAMPoints - 1) Do
   	CAM_Design.CfgIndex			:= L_CAMIndex - 1;
   	CAM_Design.V0				:= L_V2[CAM_Design.CfgIndex];
   	CAM_Design.V2				:= L_V2[L_CAMIndex];
   
   	If CAM_Design.No_Of_Points = 0 Then
   		CAM_Design.M0														:= MIO_CAM_Interface.In.Cam[L_CAMIndex - 1].Master;
   		CAM_Design.S0														:= MIO_CAM_Interface.In.Cam[L_CAMIndex - 1].Slave;
   		CAM_Design.CAM_Points[CAM_Design.No_Of_Points].Master				:= CAM_Design.M0;
   		CAM_Design.CAM_Points[CAM_Design.No_Of_Points].Slave				:= CAM_Design.S0;
   		CAM_Design.CAM_Points[CAM_Design.No_Of_Points].SegmentType			:= 1;
   		CAM_Design.No_Of_Points 											:= CAM_Design.No_Of_Points + 1;
   	Else
   		CAM_Design.M0														:= CAM_Design.CAM_Points[CAM_Design.No_Of_Points - 1].Master;
   		CAM_Design.S0														:= CAM_Design.CAM_Points[CAM_Design.No_Of_Points - 1].Slave;
   	End_If;
   
   	If L_CAMIndex = (L_NbCAMPoints - 1) Then
   		CAM_Design.V2				:= MIO_CAM_Interface.In.EndSlope;
   	Elsif ABS(CAM_Design.V2) <= 0.01 Then
   		CAM_Design.V2				:= 0;
   	End_If;
   
   	If CAM_Design.CfgIndex	 > 1 Then
   		CAM_Design.PrevSlope			:= (MIO_CAM_Interface.In.Cam[CAM_Design.CfgIndex].Slave - MIO_CAM_Interface.In.Cam[CAM_Design.CfgIndex-1].Slave) / (MIO_CAM_Interface.In.Cam[CAM_Design.CfgIndex].Master - MIO_CAM_Interface.In.Cam[CAM_Design.CfgIndex-1].Master);
   		CAM_Design.ActSlope				:= (MIO_CAM_Interface.In.Cam[CAM_Design.CfgIndex+1].Slave - MIO_CAM_Interface.In.Cam[CAM_Design.CfgIndex].Slave) / (MIO_CAM_Interface.In.Cam[CAM_Design.CfgIndex+1].Master - MIO_CAM_Interface.In.Cam[CAM_Design.CfgIndex].Master);
   	End_If;
   
   	CAM_Design.dM 					:= MIO_CAM_Interface.In.Cam[L_CAMIndex].Master - CAM_Design.M0;
   	CAM_Design.dS					:= MIO_CAM_Interface.In.Cam[L_CAMIndex].Slave - CAM_Design.S0;
   
   	If L_CAMIndex = 1 Then
   		CAM_Design.V0 				:= MIO_CAM_Interface.In.StartSlope;
   	End_If;
   
   	If (MIO_CAM_Interface.In.Cam[L_CAMIndex - 1].SegmentType = 0) Then
   		CAM_Design.CAM_Points[CAM_Design.No_Of_Points].Master				:= CAM_Design.CAM_Points[CAM_Design.No_Of_Points - 1].Master + CAM_Design.dM;
   		CAM_Design.CAM_Points[CAM_Design.No_Of_Points].Slave				:= CAM_Design.CAM_Points[CAM_Design.No_Of_Points - 1].Slave + CAM_Design.dS;
   		CAM_Design.CAM_Points[CAM_Design.No_Of_Points - 1].SegmentType		:= 0;
   		CAM_Design.CAM_Points[CAM_Design.No_Of_Points].SegmentType			:= 1;
   		CAM_Design.No_Of_Points 											:= CAM_Design.No_Of_Points + 1;
   		CAM_Design.MemoRiseReturnComp										:= 0;
   	Elsif (MIO_CAM_Interface.In.Cam[L_CAMIndex - 1].SegmentType = 1) And (MIO_CAM_Interface.In.Cfg_Segments[CAM_Design.CfgIndex].ProfilType <> 0) Then
   		AOI_PosComp_ST(L_AOI_CAM_PosComp,CAM_Design,MIO_CAM_Interface.In.Cfg_Segments);
   		If CAM_Design.Err Then
   				Sts_ERR					:= 191;
   				Sts_EXERR				:= 0;
   				Sts_ER					:= 1;
   				Sts_IP					:= 0;
   				TND();
   		End_If;
   	Elsif ((MIO_CAM_Interface.In.Cam[L_CAMIndex - 1].SegmentType = 1) And (MIO_CAM_Interface.In.Cfg_Segments[CAM_Design.CfgIndex].ProfilType = 0))  Then
   		CAM_Design.CAM_Points[CAM_Design.No_Of_Points].Master				:= CAM_Design.CAM_Points[CAM_Design.No_Of_Points - 1].Master + CAM_Design.dM;
   		CAM_Design.CAM_Points[CAM_Design.No_Of_Points].Slave				:= CAM_Design.CAM_Points[CAM_Design.No_Of_Points - 1].Slave + CAM_Design.dS;
   		CAM_Design.CAM_Points[CAM_Design.No_Of_Points - 1].SegmentType		:= 1;
   		CAM_Design.CAM_Points[CAM_Design.No_Of_Points].SegmentType			:= 1;
   		CAM_Design.No_Of_Points 											:= CAM_Design.No_Of_Points + 1;
   	End_If;
   End_For;
   
   L_MI_MCCP.FLAGS							:= 0;
   CAM_Design.MemoRiseReturnComp			:= 0;
   
   If Not MIO_CAM_Interface.Cmd.CamOrCamProfil Then
   	COP(CAM_Design.CAM_Points[0],MIO_CAM_Interface.Out.Cam[0],CAM_Design.No_Of_Points);
   	MIO_CAM_Interface.Out.NbrOfCamPoints	:= CAM_Design.No_Of_Points;
   	MIO_CAM_Interface.Out.StartSlope		:= MIO_CAM_Interface.In.StartSlope;
   	MIO_CAM_Interface.Out.EndSlope			:= CAM_Design.V2;
   	Sts_IP									:= 0;
   	Sts_PC 									:= 1;
   Else
   	MCCP(L_MI_MCCP,
   		CAM_Design.CAM_Points,
   		CAM_Design.No_Of_Points,
   		MIO_CAM_Interface.In.StartSlope,
   		CAM_Design.V2,
   		MIO_CAM_Interface.Out.CamProfil);
   	If L_MI_MCCP.DN Then
   		Sts_IP								:= 0;
   		Sts_PC 								:= 1;
   	Elsif L_MI_MCCP.ER	Then
   		Sts_IP 								:= 0;
   		Sts_ER 								:= 1;
   		Sts_ERR 							:= L_MI_MCCP.ERR;
   		Sts_EXERR 							:= L_MI_MCCP.EXERR;
   	End_If;
   End_If;
   
   GSV(CST,,CurrentValue,CST[2]);
   CycleTime := CST[2]-CST[0];
END_ROUTINE

ROUTINE Prescan   (* ladder *)
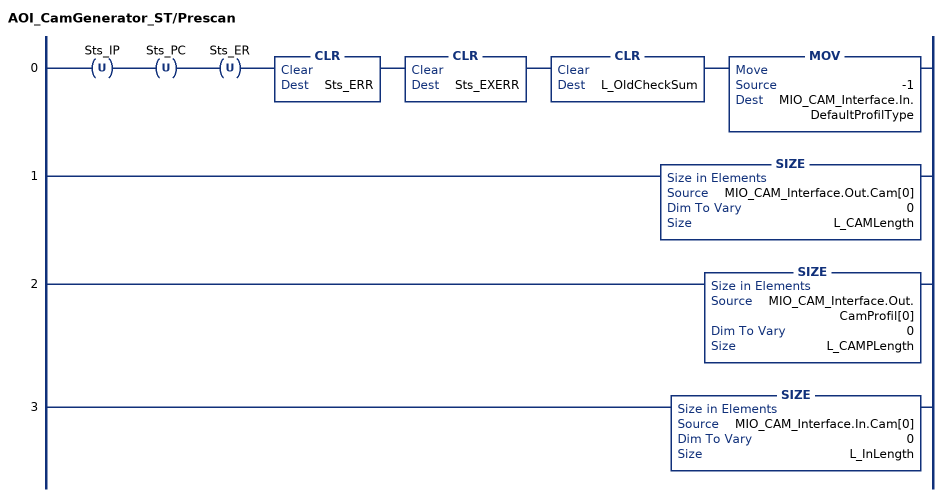
   0: OTU(Sts_IP)OTU(Sts_PC)OTU(Sts_ER)CLR(Sts_ERR)CLR(Sts_EXERR)CLR(L_OldCheckSum)MOV(-1,MIO_CAM_Interface.In.DefaultProfilType);
   1: SIZE(MIO_CAM_Interface.Out.Cam[0],0,L_CAMLength);
   2: SIZE(MIO_CAM_Interface.Out.CamProfil[0],0,L_CAMPLength);
   3: SIZE(MIO_CAM_Interface.In.Cam[0],0,L_InLength);
END_ROUTINE
END_ADD_ON_INSTRUCTION

ADD_ON_INSTRUCTION AOI_PosComp_ST   (* revision 2.0, ExecutePrescan *)
VAR_IN_OUT
   CAM_Design : UDT_CamSegment; {required}
   Cfg_Segments : UDT_SegmentSetUp[20]; {required}
END_VAR
VAR
   L_Index : REAL; {access None}
   L_Pointer : DINT; {access None}
   L_CoeffSlave : REAL[32]; {access None}
   L_CoeffMaster : REAL[32]; {access None}
   L_RawIndex : DINT; {access None}
   L_No_PtSeg : DINT; {access None}
   L_MemoCheckSum : DINT; {access None}
   L_Coeff : REAL[4]; {access None}
   L_PI : REAL; {access None}
   L_Peak : REAL; {access None}
   L_CoeffPeak : REAL[32]; {access None}
   L_Cv : REAL[2]; {access None}
   L_Mn : REAL[2]; {access None}
   L_Sn : REAL[2]; {access None}
   L_CheckSum : DINT; {access None}
   L_dV0 : REAL; {access None}
   L_NoDwell : BOOL; {access None}
   L_AccelProportion : REAL; {access None}
   L_DecelProportion : REAL; {access None}
   L_dV1 : REAL; {access None}
   L_An : REAL; {access None}
   L_M2 : REAL; {access None}
END_VAR

ROUTINE Logic   (* structured text *)
   L_CheckSum	:= CAM_Design.NbPoints + Cfg_Segments[CAM_Design.CfgIndex].ProfilType;
   
   //Compute Coeff function of selected law
   If ( L_CheckSum <> L_MemoCheckSum) Then
   	L_Index 														:= 0;
   	L_Peak															:= 0;
   	L_No_PtSeg														:= (CAM_Design.NbPoints/2);
   	L_MemoCheckSum 													:= L_CheckSum;
   
   	Case Cfg_Segments[CAM_Design.CfgIndex].ProfilType Of
   
   	2:	For L_Pointer := 1 to L_No_PtSeg do
   			L_Index 												:= L_Index + (0.5/L_No_PtSeg);
   			L_Peak 													:= L_Peak + (0.375/L_No_PtSeg);
   			If L_Index <= (1/8) Then
   				L_CoeffSlave[L_Pointer] 							:= 2/(2+L_PI)*(L_Index-0.25/L_PI*SIN(4*L_PI*L_Index));
   			Elsif (L_Index > (1/8)) And (L_Index <= (3/8)) Then
   				L_CoeffSlave[L_Pointer] 							:= 1/(2+L_PI)*(4*L_PI*(L_Index)**2+(2-L_PI)*L_Index+(L_PI**2-8)/16/L_PI);
   			Elsif (L_Index > (3/8)) And (L_Index <= (0.5)) Then
   				L_CoeffSlave[L_Pointer] 							:= 2/(2+L_PI)*((L_PI+1)*L_Index-1/4/L_PI*SIN(4*L_PI*(L_Index-1/4))-L_PI/4);
   			Elsif (L_Index > (0.5)) And (L_Index <= (5/8)) Then
   				L_CoeffSlave[L_Pointer] 							:= 1-2/(2+L_PI)*((L_PI+1)*(1-L_Index)-1/4/L_PI*SIN(4*L_PI*((1-L_Index)-1/4))-L_PI/4);
   			Elsif (L_Index > (5/8)) And (L_Index <= (7/8)) Then
   				L_CoeffSlave[L_Pointer] 							:= 1-1/(L_PI+2)*(4*L_PI*(1-L_Index)**2+(2-L_PI)*(1-L_Index)+(L_PI**2-8)/16/L_PI);
   			Else
   				L_CoeffSlave[L_Pointer] 							:= 1-2/(L_PI+2)*((1-L_Index)-1/4/L_PI*SIN(4*L_PI*(1-L_Index)));
   			End_If;
   			L_CoeffPeak[L_Pointer] 									:= L_CoeffSlave[L_Pointer]-0.017668661-0.38897*L_Peak;
   			L_CoeffMaster[L_Pointer] 								:= L_CoeffMaster[L_Pointer - 1] + (1/L_No_PtSeg);
   		End_For;
   		L_Cv[0]														:= 2;
   		L_Mn[0]														:= 0.5;
   		L_Sn[0] 													:= 0.5;
   		L_Cv[1]														:= 1.6103;
   		L_Mn[1]														:= 0.375;
   		L_Sn[1] 													:= 0.33646;
   		L_An														:= 4.88812;
   
   	3:	L_No_PtSeg													:= 5;
   		For L_Pointer := 1 to L_No_PtSeg do
   			L_Index 												:= L_Index + 0.25;
   			L_Peak 													:= L_Index;
   			L_CoeffSlave[L_Pointer] 								:= 3*((L_Index)**2) - 2*((L_Index)**3);
   			L_CoeffPeak[L_Pointer] 									:= L_CoeffSlave[L_Pointer];
   			L_CoeffMaster[L_Pointer] 								:= L_CoeffMaster[L_Pointer - 1] + 0.5;
   		End_For;
   		L_No_PtSeg													:= 2;
   		L_Cv[0]														:= 1.5;
   		L_Mn[0]														:= 0.5;
   		L_Sn[0] 													:= 0.5;
   		L_Cv[1]														:= 1.5;
   		L_Mn[1]														:= 0.5;
   		L_Sn[1] 													:= 0.5;
   		L_An														:= 4;
   
   	4:	For L_Pointer := 1 to L_No_PtSeg do
   			L_Index 												:= L_Index + (0.5/L_No_PtSeg);
   			L_Peak 													:= L_Peak + (0.374974995022058/L_No_PtSeg);
   			If L_Index < (1/8) Then
   				L_CoeffSlave[L_Pointer] 							:= L_PI/(4+L_PI)*(L_Index-1/4/L_PI*SIN(4*L_PI*L_Index));
   			Else
   				L_CoeffSlave[L_Pointer] 							:= L_PI/(4+L_PI)*(2/L_PI+L_Index-9/4/L_PI*SIN(L_PI/3*(1+4*L_Index)));
   			End_If;
   			If (L_Peak+0.125025004977942) < (1/8) Then
   				L_CoeffPeak[L_Pointer] 								:= L_PI/(4+L_PI)*((L_Peak+0.125025004977942)-1/4/L_PI*SIN(4*L_PI*(L_Peak+0.125025004977942)))-0.0199924101557209-0.440039072926203*L_Peak;
   			Else
   				L_CoeffPeak[L_Pointer] 								:= L_PI/(4+L_PI)*(2/L_PI+(L_Peak+0.125025004977942)-9/4/L_PI*SIN(L_PI/3*(1+4*(L_Peak+0.125025004977942))))-0.0199924101557209-0.440039072926203*L_Peak;
   			End_If;
   			L_CoeffMaster[L_Pointer] 								:= L_CoeffMaster[L_Pointer - 1] + (1/L_No_PtSeg);
   		End_For;
   		L_Cv[0]														:= 1.7596;
   		L_Mn[0]														:= 0.5;
   		L_Sn[0] 													:= 0.5;
   		L_Cv[1]														:= 1.3195609270738;
   		L_Mn[1]														:= 0.374974995022058;
   		L_Sn[1] 													:= 0.315003940664265;
   		L_An														:= 5.527957357;
   
   	5:	For L_Pointer := 1 to L_No_PtSeg do
   			L_Index 												:= L_Index + (0.5/L_No_PtSeg);
   			L_CoeffSlave[L_Pointer] 								:= 6*((L_Index)**5) - 15*((L_Index)**4) + 10*((L_Index)**3);
   			L_Peak													:= L_Peak + (0.288657731551211/L_No_PtSeg);
   			L_CoeffPeak[L_Pointer]									:= 6*((L_Peak+0.211342268448789)**5) - 15*((L_Peak+0.211342268448789)**4) + 10*((L_Peak+0.211342268448789)**3)-(0.833433809852203*L_Peak)-0.0670018015184139;
   			L_CoeffMaster[L_Pointer] 								:= L_CoeffMaster[L_Pointer - 1] + (1/L_No_PtSeg);
   		End_For;
   		L_Cv[0]														:= 1.875;
   		L_Mn[0]														:= 0.5;
   		L_Sn[0] 													:= 0.5;
   		L_Cv[1]														:= 1.0415661901478;
   		L_Mn[1]														:= 0.288657731551211;
   		L_Sn[1] 													:= 0.192421085531565;
   		L_An														:= 5.77350283926745;
   
   	7:	For L_Pointer := 1 to L_No_PtSeg do
   			L_Index 												:= L_Index + (0.5/L_No_PtSeg);
   			L_CoeffSlave[L_Pointer] 								:= 35*((L_Index)**4) - 84*((L_Index)**5) + 70*((L_Index)**6) - 20*((L_Index)**7);
   			L_Peak			 										:= L_Peak + (0.223644728961517/L_No_PtSeg);
   			L_CoeffPeak[L_Pointer]									:= 35*(L_Peak+0.276355271038483)**4-84*(L_Peak+0.276355271038483)**5+70*(L_Peak+0.276355271038483)**6-20*(L_Peak+0.276355271038483)**7-0.0974652864980157-1.11971501566437*L_Peak;
   			L_CoeffMaster[L_Pointer] 								:= L_CoeffMaster[L_Pointer - 1] + (1/L_No_PtSeg);
   		End_For;
   		L_Cv[0]														:= 2.19;
   		L_Mn[0]														:= 0.5;
   		L_Sn[0] 													:= 0.5;
   		L_Cv[1]														:= 1.07028498433563;
   		L_Mn[1]														:= 0.223644728961517;
   		L_Sn[1] 													:= 0.152116352309586;
   		L_An														:= 7.513188448;
   
   	Else
   		CAM_Design.Err												:= 1;
   		TND();
   	End_Case;
   End_If;
   
   If CAM_Design.RiseReturnComp[CAM_Design.CfgIndex] And Not CAM_Design.MemoRiseReturnComp Then
   	L_Coeff[0]														:= ((1/L_Cv[0])/L_Mn[0]);
   	L_Coeff[1]														:= ((1/L_Cv[1])/L_Mn[1]);
   	L_Coeff[2]														:= L_Coeff[0]*L_Sn[0];
   	L_Coeff[3]														:= L_Coeff[1]*L_Sn[1];
   Elsif CAM_Design.MemoRiseReturnComp And Not CAM_Design.RiseReturnComp[CAM_Design.CfgIndex] Then
   	L_Coeff[0]														:= ((1/L_Cv[1])/L_Mn[1]);
   	L_Coeff[1]														:= ((1/L_Cv[0])/L_Mn[0]);
   	L_Coeff[2]														:= L_Coeff[0]*L_Sn[1];
   	L_Coeff[3]														:= L_Coeff[1]*L_Sn[0];
   Elsif CAM_Design.MemoRiseReturnComp And CAM_Design.RiseReturnComp[CAM_Design.CfgIndex] Then
   	L_Coeff[0]														:= ((1/L_Cv[1])/L_Mn[1]);
   	L_Coeff[1]														:= L_Coeff[0];
   	L_Coeff[2]														:= L_Coeff[0]*L_Sn[1];
   	L_Coeff[3]														:= L_Coeff[2];
   Else
   	L_Coeff[0]														:= ((1/L_Cv[0])/L_Mn[0]);
   	L_Coeff[1]														:= L_Coeff[0];
   	L_Coeff[2]														:= L_Coeff[0]*L_Sn[0];
   	L_Coeff[3]														:= L_Coeff[2];
   End_If;
   
   //Estimate velocity
   If CAM_Design.V0 <> CAM_Design.V2 Then
   	CAM_Design.V1													:= ((((CAM_Design.dS - (CAM_Design.dM * CAM_Design.V0)) - ((CAM_Design.V2 - CAM_Design.V0) * (CAM_Design.dM/2) * (1 - L_Coeff[3]))) / (((CAM_Design.dM/2)*L_Coeff[2]) + ((CAM_Design.dM/2)*L_Coeff[3])))) + CAM_Design.V0;
   Else
   	CAM_Design.V1													:= (CAM_Design.dS / CAM_Design.dM) * (L_Cv[0]/L_Cv[1]);
   End_If;
   
   If CAM_Design.MemoRiseReturnComp Then
   	If ABS(CAM_Design.ActSlope) = ABS(CAM_Design.PrevSlope) Then
   		L_AccelProportion											:= Cfg_Segments[CAM_Design.CfgIndex-1].DecelProportion;
   		L_DecelProportion											:= Cfg_Segments[CAM_Design.CfgIndex-1].AccelProportion;
   	Else
   		L_M2														:= ABS(CAM_Design.V1 / CAM_Design.a4)* ((L_An/L_Cv[1])*L_Mn[1]);//(L_Cv[1]+L_Mn[1]);
   		L_AccelProportion											:= CAM_Design.dM/L_M2;
   		L_DecelProportion											:= CAM_Design.dM/(CAM_Design.dM - L_M2);
   		If L_AccelProportion <= 1 Then
   			If ABS(CAM_Design.a4) < 0.01 Then
   				L_AccelProportion									:= 2;
   				L_DecelProportion 									:= 2;
   				CAM_Design.MemoRiseReturnComp						:= 0;
   				If CAM_Design.RiseReturnComp[CAM_Design.CfgIndex] Then
   					L_Coeff[0]										:= ((1/L_Cv[0])/L_Mn[0]);
   					L_Coeff[1]										:= ((1/L_Cv[1])/L_Mn[1]);
   					L_Coeff[2]										:= L_Coeff[0]*L_Sn[0];
   					L_Coeff[3]										:= L_Coeff[1]*L_Sn[1];
   				Else
   					L_Coeff[0]										:= ((1/L_Cv[0])/L_Mn[0]);
   					L_Coeff[1]										:= L_Coeff[0];
   					L_Coeff[2]										:= L_Coeff[0]*L_Sn[0];
   					L_Coeff[3]										:= L_Coeff[2];
   				End_If;
   			Else
   				L_AccelProportion									:= 3/2;
   				L_DecelProportion 									:= 3;
   			End_If;
   		End_If;
   	End_If;
   Else
   	L_AccelProportion												:= Cfg_Segments[CAM_Design.CfgIndex].AccelProportion;
   	L_DecelProportion												:= Cfg_Segments[CAM_Design.CfgIndex].DecelProportion;
   End_If;
   
   If (L_AccelProportion <= 0) And (L_DecelProportion <= 0) Then
   	CAM_Design.M2													:= CAM_Design.dM/3;
   	CAM_Design.M4													:= CAM_Design.M2  ;
   	L_NoDwell														:= 0;
   Elsif ((L_AccelProportion > 0) And (L_DecelProportion > 0)
   And (L_AccelProportion <> 1) And (L_DecelProportion <> 1)) Then
   	CAM_Design.M2													:= (CAM_Design.dM / L_AccelProportion);
   	CAM_Design.M4													:= (CAM_Design.dM / L_DecelProportion);
   	CAM_Design.K2													:= CAM_Design.M2 + CAM_Design.M4;
   	L_NoDwell														:= 0;
   	If (CAM_Design.K2 >= CAM_Design.dM) Then
   		CAM_Design.M2												:= (CAM_Design.dM / L_AccelProportion);
   		CAM_Design.M4												:= (CAM_Design.dM - CAM_Design.M2);
   		L_NoDwell													:= 1;
   	End_If;
   Elsif (L_AccelProportion > 0) And (L_DecelProportion <= 0)
   And (L_AccelProportion <> 1) Then
   	CAM_Design.M2													:= (CAM_Design.dM / L_AccelProportion);
   	CAM_Design.M4													:= (CAM_Design.dM - CAM_Design.M2);
   	L_NoDwell														:= 1;
   Elsif (L_AccelProportion <= 0) And (L_DecelProportion > 0)
   And (L_DecelProportion <> 1) Then
   	CAM_Design.M4													:= (CAM_Design.dM / L_DecelProportion);
   	CAM_Design.M2													:= (CAM_Design.dM - CAM_Design.M4);
   	L_NoDwell														:= 1;
   Elsif (L_AccelProportion = 1) Or (L_DecelProportion = 1) Then
   	CAM_Design.M2													:= (CAM_Design.dM / 2);
   	CAM_Design.M4													:= CAM_Design.M2;
   	L_NoDwell														:= 1;
   End_If;
   
   CAM_Design.M3														:= CAM_Design.dM -(CAM_Design.M2 + CAM_Design.M4);
   
   CAM_Design.K2														:= (CAM_Design.M2*L_Coeff[2]) + CAM_Design.M3 + (CAM_Design.M4*L_Coeff[3]);
   If CAM_Design.K2 <= 0 Then
   	CAM_Design.Err													:= 1;
   	TND();
   Else
   	CAM_Design.V1													:= (((CAM_Design.dS - (CAM_Design.dM * CAM_Design.V0)) - ((CAM_Design.V2 - CAM_Design.V0) * CAM_Design.M4 * (1 - L_Coeff[3]))) / CAM_Design.K2) + CAM_Design.V0;
   	CAM_Design.K1													:= (CAM_Design.V1 - CAM_Design.V0) * CAM_Design.M2 * L_Coeff[0];
   	CAM_Design.K5													:= (CAM_Design.V1 - CAM_Design.V2) * CAM_Design.M4 * L_Coeff[1];
   	CAM_Design.S3													:= CAM_Design.M3 * CAM_Design.V1;
   End_If;
   
   For L_RawIndex := 1 to L_No_PtSeg Do
   	CAM_Design.K3													:= L_CoeffMaster[L_RawIndex] * CAM_Design.M2;
   	CAM_Design.CAM_Points[CAM_Design.No_Of_Points].Master 			:= CAM_Design.M0 + CAM_Design.K3;
   	If CAM_Design.MemoRiseReturnComp Then
   		CAM_Design.CAM_Points[CAM_Design.No_Of_Points].Slave 		:= (CAM_Design.V0 * CAM_Design.K3) + (L_CoeffPeak[L_RawIndex] * CAM_Design.K1) + CAM_Design.S0;
   	Else
   		CAM_Design.CAM_Points[CAM_Design.No_Of_Points].Slave 		:= (CAM_Design.V0 * CAM_Design.K3) + (L_CoeffSlave[L_RawIndex] * CAM_Design.K1) + CAM_Design.S0;
   	End_If;
   	CAM_Design.CAM_Points[CAM_Design.No_Of_Points].SegmentType 		:= 1;
   	CAM_Design.No_Of_Points 										:= CAM_Design.No_Of_Points + 1;
   End_For;
   If CAM_Design.MemoRiseReturnComp Then
   	CAM_Design.MemoRiseReturnComp									:= 0;
   End_If;
   
   CAM_Design.M5 														:= CAM_Design.CAM_Points[CAM_Design.No_Of_Points - 1].Master + CAM_Design.M3;
   CAM_Design.S5 														:= CAM_Design.CAM_Points[CAM_Design.No_Of_Points - 1].Slave + CAM_Design.S3;
   If Not L_NoDwell And (CAM_Design.M3 > 0.1) Then
   	CAM_Design.CAM_Points[CAM_Design.No_Of_Points].Master 			:= CAM_Design.M5;
   	CAM_Design.CAM_Points[CAM_Design.No_Of_Points].Slave 			:= CAM_Design.S5;
   	CAM_Design.CAM_Points[CAM_Design.No_Of_Points].SegmentType 		:= 1;
   	CAM_Design.CAM_Points[CAM_Design.No_Of_Points - 1].SegmentType 	:= 0;
   	CAM_Design.No_Of_Points 										:= CAM_Design.No_Of_Points + 1;
   End_If;
   
   For L_RawIndex := 1 to L_No_PtSeg Do
   	CAM_Design.K3													:= L_CoeffMaster[L_RawIndex] * CAM_Design.M4;
   	CAM_Design.CAM_Points[CAM_Design.No_Of_Points].Master 			:= CAM_Design.M5 + CAM_Design.K3;
   	If CAM_Design.RiseReturnComp[CAM_Design.CfgIndex] Then
   		CAM_Design.CAM_Points[CAM_Design.No_Of_Points].Slave 		:= (CAM_Design.V2 * CAM_Design.K3) + ((L_Sn[1] - L_CoeffPeak[L_No_PtSeg - L_RawIndex]) * CAM_Design.K5) + CAM_Design.S5;
   	Else
   		CAM_Design.CAM_Points[CAM_Design.No_Of_Points].Slave 		:= (CAM_Design.V2 * CAM_Design.K3) + ((L_Sn[0] - L_CoeffSlave[L_No_PtSeg - L_RawIndex]) * CAM_Design.K5) + CAM_Design.S5;
   	End_If;
   	CAM_Design.CAM_Points[CAM_Design.No_Of_Points].SegmentType 		:= 1;
   	CAM_Design.No_Of_Points 										:= CAM_Design.No_Of_Points + 1;
   End_For;
   If CAM_Design.RiseReturnComp[CAM_Design.CfgIndex] Then
   	CAM_Design.MemoRiseReturnComp									:= 1;
   End_If;
   
   CAM_Design.CAM_Points[CAM_Design.No_Of_Points-1].Master 			:= CAM_Design.dM + CAM_Design.M0;
   CAM_Design.CAM_Points[CAM_Design.No_Of_Points-1].Slave 				:= CAM_Design.dS + CAM_Design.S0;
   
   CAM_Design.a4 														:= ((CAM_Design.V2 - CAM_Design.V1) / CAM_Design.M4)*((L_An/L_Cv[1])*L_Mn[1]);
END_ROUTINE

ROUTINE Prescan   (* ladder *)
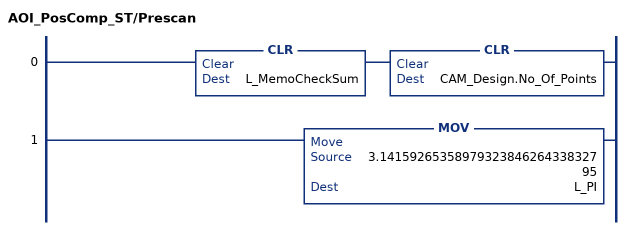
   0: CLR(L_MemoCheckSum)CLR(CAM_Design.No_Of_Points);
   1: MOV(3.1415926535897932384626433832795,L_PI);
END_ROUTINE
END_ADD_ON_INSTRUCTION

ADD_ON_INSTRUCTION Axis_speed_control   (* revision 2.0 *)
VAR_IN_OUT
   Axis : AXIS_CIP_DRIVE; {required}
END_VAR
VAR_INPUT
   Enable : BOOL; {required}
   Speed : REAL; {required}
   Acc : REAL; {required}
   Dec : REAL; {required}
   Jerk : REAL; {required}
END_VAR
VAR_OUTPUT
   IP : BOOL; {access Read Only, visible}
   ER : BOOL; {access Read Only, visible}
END_VAR
VAR
   MASR_AXE : MOTION_INSTRUCTION;
   MAFR_AXE : MOTION_INSTRUCTION;
   MAS_AXE : MOTION_INSTRUCTION;
   MCD_Jog : MOTION_INSTRUCTION;
   erreur_1 : BOOL;
   erreur_2 : BOOL;
   Speed_direction : REAL;
   MAS_Jog : MOTION_INSTRUCTION; {access None}
   MAJ_Jog : MOTION_INSTRUCTION; {access None}
   MSO_Test : MOTION_INSTRUCTION; {access None}
   MSF_Test : MOTION_INSTRUCTION; {access None}
END_VAR

ROUTINE Logic   (* ladder *)
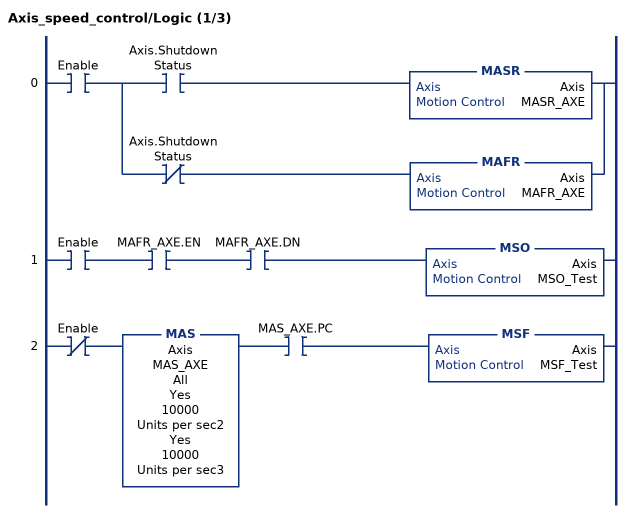
   0: XIC(Enable)[XIC(Axis.ShutdownStatus) MASR(Axis,MASR_AXE) ,XIO(Axis.ShutdownStatus) MAFR(Axis,MAFR_AXE) ];
   1: XIC(Enable)XIC(MAFR_AXE.EN)XIC(MAFR_AXE.DN)MSO(Axis,MSO_Test);
   2: XIO(Enable)MAS(Axis,MAS_AXE,All,Yes,10000,Units per sec2,Yes,10000,Units per sec3)XIC(MAS_AXE.PC)MSF(Axis,MSF_Test);
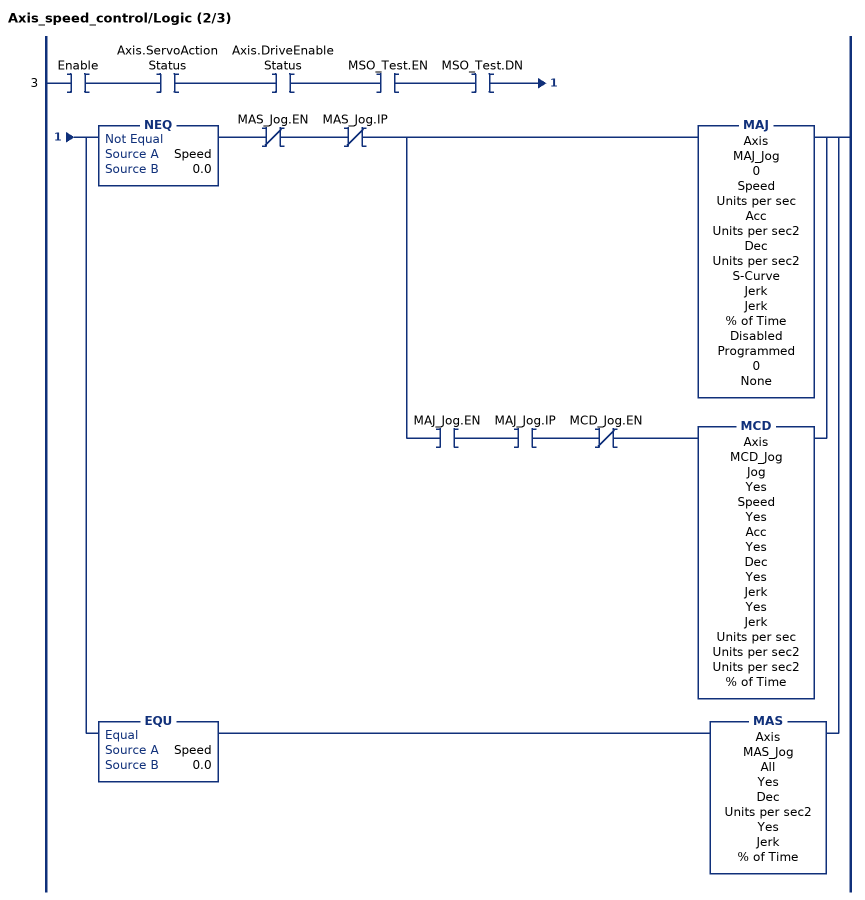
   3: XIC(Enable)XIC(Axis.ServoActionStatus)XIC(Axis.DriveEnableStatus)XIC(MSO_Test.EN)XIC(MSO_Test.DN)[NEQ(Speed,0.0) XIO(MAS_Jog.EN) XIO(MAS_Jog.IP) [MAJ(Axis,MAJ_Jog,0,Speed,Units per sec,Acc,Units per sec2,Dec,Units per sec2,S-Curve,Jerk,Jerk,% of Time,Disabled,Programmed,0,None) ,XIC(MAJ_Jog.EN) XIC(MAJ_Jog.IP) XIO(MCD_Jog.EN) MCD(Axis,MCD_Jog,Jog,Yes,Speed,Yes,Acc,Yes,Dec,Yes,Jerk,Yes,Jerk,Units per sec,Units per sec2,Units per sec2,% of Time) ] ,EQU(Speed,0.0) MAS(Axis,MAS_Jog,All,Yes,Dec,Units per sec2,Yes,Jerk,% of Time) ];
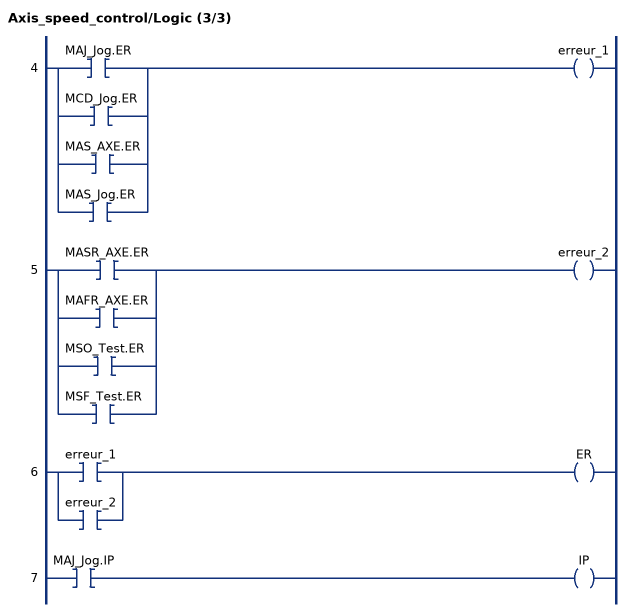
   4: [XIC(MAJ_Jog.ER) ,XIC(MCD_Jog.ER) ,XIC(MAS_AXE.ER) ,XIC(MAS_Jog.ER) ]OTE(erreur_1);
   5: [XIC(MASR_AXE.ER) ,XIC(MAFR_AXE.ER) ,XIC(MSO_Test.ER) ,XIC(MSF_Test.ER) ]OTE(erreur_2);
   6: [XIC(erreur_1) ,XIC(erreur_2) ]OTE(ER);
   7: XIC(MAJ_Jog.IP)OTE(IP);
END_ROUTINE
END_ADD_ON_INSTRUCTION

ADD_ON_INSTRUCTION Badges_Acces   (* revision 1.2 *)
// Revision note:
// V1.0: GUY: Version initiale
// V1.1: ROD: Modification pour login distant
// V1.2: GUY: Debug login distant
VAR_INPUT
   Lecteur_Badge_Code_A : BOOL; {required}
   Lecteur_Badge_Code_B : BOOL; {required}
   Lecteur_Badge_Code_C : BOOL; {required}
   Lecteur_Badge_Code_D : BOOL; {required}
END_VAR
VAR_OUTPUT
   Badge_Code_A : BOOL; {required}
   Badge_Code_B : BOOL; {required}
   Badge_Code_C : BOOL; {required}
   Badge_Code_D : BOOL; {required}
   Badge_Temps_Restant : DINT; {required}
END_VAR
VAR_INPUT
   Badge_RAZ_Code : BOOL; {required}
   Tempo_Logout_1 : DINT; {required}
   Tempo_Logout_2 : DINT; {required}
   Tempo_Logout_3 : DINT; {required}
END_VAR
VAR
   Badge_code_en_cours : BOOL;
   Badge_Tempo_Logout : TIMER := (PRE := 600000);
   Tempo_Logout_Utilisee : DINT := 600000;
   Front_Badge_Code_A : BOOL;
   Front_Badge_Code_A_temp : BOOL;
   Front_Badge_Code_B : BOOL;
   Front_Badge_Code_B_temp : BOOL;
   Front_Badge_Code_C : BOOL;
   Front_Badge_Code_C_temp : BOOL;
   Front_Badge_Code_D : BOOL;
   Front_Badge_Code_D_temp : BOOL;
   Front_Raz_Badge : BOOL; {access None}
   Tempo_Forcage_Code_D : TIMER; {access None}
END_VAR

ROUTINE Logic   (* ladder *)
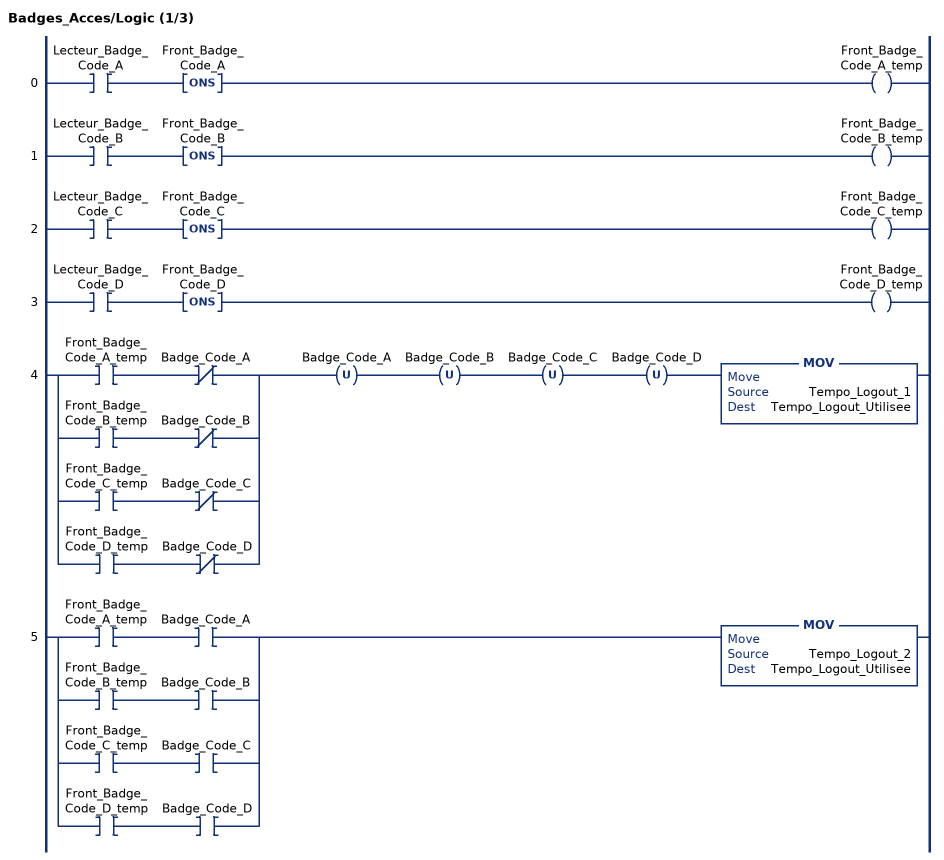
   0: XIC(Lecteur_Badge_Code_A)ONS(Front_Badge_Code_A)OTE(Front_Badge_Code_A_temp);
   1: XIC(Lecteur_Badge_Code_B)ONS(Front_Badge_Code_B)OTE(Front_Badge_Code_B_temp);
   2: XIC(Lecteur_Badge_Code_C)ONS(Front_Badge_Code_C)OTE(Front_Badge_Code_C_temp);
   3: XIC(Lecteur_Badge_Code_D)ONS(Front_Badge_Code_D)OTE(Front_Badge_Code_D_temp);
   4: [XIC(Front_Badge_Code_A_temp) XIO(Badge_Code_A) ,XIC(Front_Badge_Code_B_temp) XIO(Badge_Code_B) ,XIC(Front_Badge_Code_C_temp) XIO(Badge_Code_C) ,XIC(Front_Badge_Code_D_temp) XIO(Badge_Code_D) ]OTU(Badge_Code_A)OTU(Badge_Code_B)OTU(Badge_Code_C)OTU(Badge_Code_D)MOV(Tempo_Logout_1,Tempo_Logout_Utilisee);
   5: [XIC(Front_Badge_Code_A_temp) XIC(Badge_Code_A) ,XIC(Front_Badge_Code_B_temp) XIC(Badge_Code_B) ,XIC(Front_Badge_Code_C_temp) XIC(Badge_Code_C) ,XIC(Front_Badge_Code_D_temp) XIC(Badge_Code_D) ]MOV(Tempo_Logout_2,Tempo_Logout_Utilisee);
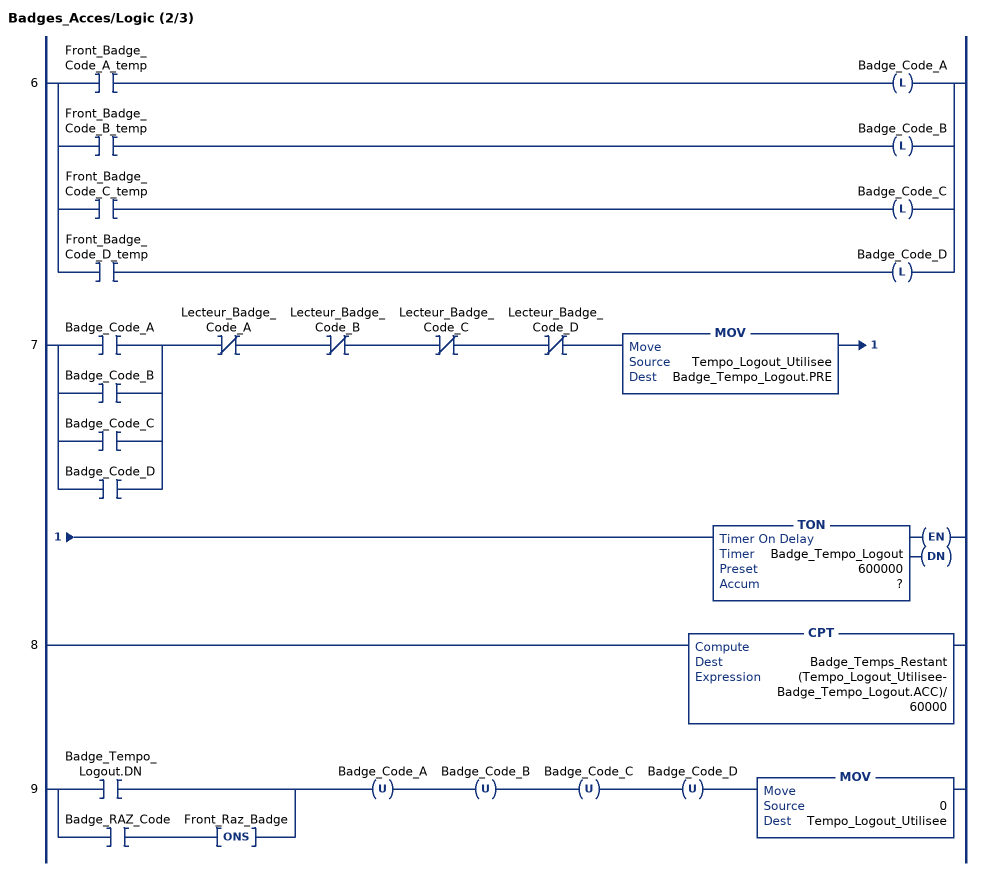
   6: [XIC(Front_Badge_Code_A_temp) OTL(Badge_Code_A) ,XIC(Front_Badge_Code_B_temp) OTL(Badge_Code_B) ,XIC(Front_Badge_Code_C_temp) OTL(Badge_Code_C) ,XIC(Front_Badge_Code_D_temp) OTL(Badge_Code_D) ];
   7: [XIC(Badge_Code_A) ,XIC(Badge_Code_B) ,XIC(Badge_Code_C) ,XIC(Badge_Code_D) ]XIO(Lecteur_Badge_Code_A)XIO(Lecteur_Badge_Code_B)XIO(Lecteur_Badge_Code_C)XIO(Lecteur_Badge_Code_D)MOV(Tempo_Logout_Utilisee,Badge_Tempo_Logout.PRE)TON(Badge_Tempo_Logout,?,?);
   8: CPT(Badge_Temps_Restant,(Tempo_Logout_Utilisee-Badge_Tempo_Logout.ACC)/60000);
   9: [XIC(Badge_Tempo_Logout.DN) ,XIC(Badge_RAZ_Code) ONS(Front_Raz_Badge) ]OTU(Badge_Code_A)OTU(Badge_Code_B)OTU(Badge_Code_C)OTU(Badge_Code_D)MOV(0,Tempo_Logout_Utilisee);
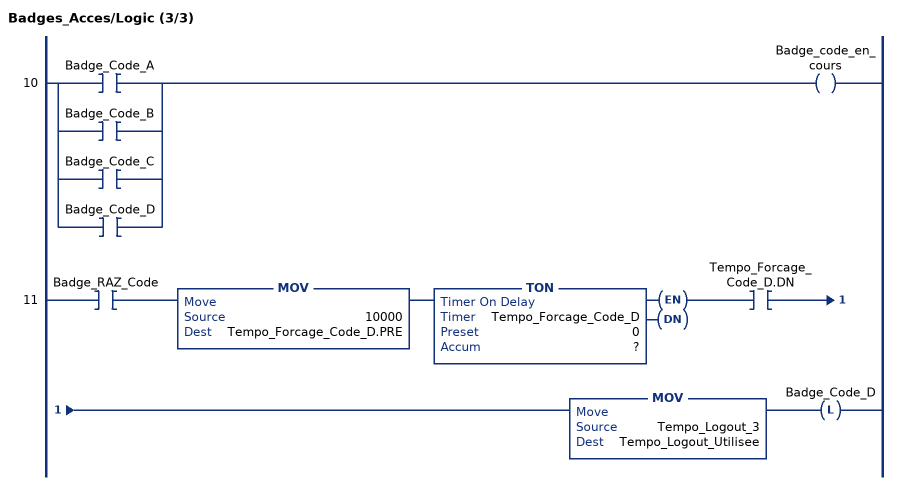
   10: [XIC(Badge_Code_A) ,XIC(Badge_Code_B) ,XIC(Badge_Code_C) ,XIC(Badge_Code_D) ]OTE(Badge_code_en_cours);
   11: XIC(Badge_RAZ_Code)MOV(10000,Tempo_Forcage_Code_D.PRE)TON(Tempo_Forcage_Code_D,?,?)XIC(Tempo_Forcage_Code_D.DN)MOV(Tempo_Logout_3,Tempo_Logout_Utilisee)OTL(Badge_Code_D);
END_ROUTINE
END_ADD_ON_INSTRUCTION

ADD_ON_INSTRUCTION Engage_Axe   (* revision 1.14 *)
// Revision note:
// v1.14: Modification Changement de Came en Synchro
// v1.13: Modification phase Vnul
// v1.12: Ajout de retour d'engagement
// v1.11: Ajout changement de came
// v1.10: Ajout des zones de changement de came
// v1.9: Correction Bug maitre à l'arret dans zone d'embrayage: (L16)
//    - Optimisation avec pending status
//    - Forward Only / Bi direc sur MAPC
//    - Command pos au lieu de actual pos sur MAPC
// v1.8: Lancement de came en mode Once (L17)
// v1.7: Degagemennt en position sur front (L8)
VAR_IN_OUT
   Axe : AXIS_CIP_DRIVE; {required}   // Axe esclave a controler
   Axe_Maitre : AXIS_VIRTUAL; {required}   // Axe maitre de la came
END_VAR
VAR_INPUT
   Activation : BOOL; {required}   // Activation puissance A Activer avant d'engager
   Engagement : BOOL; {required}   // Engagement de l'axe sur profil de came
   Maitre_V_Nul : BOOL; {required}   // Engagement avec Maitre vitesse nul (positionnement à l'arret)
   Engagement_Decalage : BOOL; {required}   // Activation du decalage en marche
   Degagement_en_pos : BOOL; {required}   // Attente position pour degagement
   Val_Vitesse : REAL; {required}   // Valeur de vitesse global de l'axe
   Val_Acc : REAL; {required}   // Valeur d accel gloable de laxe
   Val_Dec : REAL; {required}   // Valeur de decel
   Val_Jerk : REAL; {required}   // Valeur de jerk
   Val_Engagement : REAL; {required}   // Valeur Absolu d'engagement (0 ou 1 pour axe rotatif)
   Val_Degagement : REAL; {required}   // Valeur de degagement de l'axe (0 ou 1 pour axe rotatif)
   Val_Phase : REAL; {required}   // Valeur de Phase
   Val_Decalage : REAL; {required}   // Valeur de decalage (actif si bit d'activation a 1)
END_VAR
VAR_IN_OUT
   Came : CAM[100]; {required}   // Came modifiable a la volée (tableau de la came)
END_VAR
VAR_INPUT
   Longeur_Cam : DINT; {required}   // Longeur de la came (doit etre sup a 3)
   Modulo_Maitre : REAL; {required}   // Longeur du maitre pour calcul de la phase (modulo maitre)
   Mode_Rotatif : BOOL; {required}   // Activation mode rotatif (MAM type 2 au lieu de 0 pour le pre positionnement)
   Modulo_Esclave : DINT; {required}   // Utilise seulement pour engagement a vnul et rotatif (valeur du modulo de l'axe rotatif)
END_VAR
VAR_OUTPUT
   Axe_Engage : BOOL; {access Read Only, visible}   // Axe engage sur came
   Axe_Degage : BOOL; {access Read Only, visible}   // Axe Degage
   ER : BOOL; {access Read Only, visible}   // Erreur dans le module (retour des blocs fonction)
END_VAR
VAR_INPUT
   Num_Cam_Vnul : DINT;
   ModeCamOnce : BOOL; {required}   // Came en mode once (actif = 1)
   Top_Once : BOOL; {required}   // Top de lancement en mode once
   Start_Slope : REAL; {access None, required}
   Stop_Slope : REAL; {access None, required}
END_VAR
VAR_OUTPUT
   Changement_Came_Actif : BOOL; {access None, visible}
   Preposition_OK : BOOL; {access Read Only, visible}
END_VAR
VAR
   MSO_desactivation : MOTION_INSTRUCTION;
   MSO_activation : MOTION_INSTRUCTION;
   MAS_degagement : MOTION_INSTRUCTION;
   MAS_Engagement : MOTION_INSTRUCTION;
   MCCP_1 : MOTION_INSTRUCTION;
   Came_Prof_1 : CAM_PROFILE[100];
   MAPC_1 : MOTION_INSTRUCTION;
   Front : BOOL;
   Val_Phase_Sauve : REAL;
   Val_Phase_Modifie : REAL;
   MAM_Phase : MOTION_INSTRUCTION;
   Engagement_came : BOOL;
   MAM_decalage : MOTION_INSTRUCTION;
   MCCP_2 : MOTION_INSTRUCTION;
   MCCP_First : MOTION_INSTRUCTION;
   MAPC_First : MOTION_INSTRUCTION;
   Came_Prof_2 : CAM_PROFILE[100];
   Came_Prof_First : CAM_PROFILE[100];
   MAPC_2 : MOTION_INSTRUCTION;
   Top_Calage0 : BOOL;
   TEMP_0 : BOOL;
   TEMP_1 : BOOL;
   Top_Calage1 : BOOL;
   Axe_Active : BOOL;
   Num_Cam : DINT;
   Val_phase_modulo : REAL;
   Erreur_1 : BOOL;
   Erreur_2 : BOOL;
   MAS_degagement_enpos : MOTION_INSTRUCTION;
   DEGagement_En_Pos_ok : BOOL;
   Top_Calage2 : BOOL;
   TEMP_2 : BOOL;
   TEMP_3 : BOOL;
   Top_Calage3 : BOOL;
   Val_Engagement_plus : REAL;
   MAM_degagement_rotatif : MOTION_INSTRUCTION;
   MAM_degagement_lineaire : MOTION_INSTRUCTION;
   MAM_degagement_enpos_lineaire : MOTION_INSTRUCTION;
   MAM_degagement_enpos_rotatif : MOTION_INSTRUCTION;
   MAM_engagement_rotatif : MOTION_INSTRUCTION;
   MAM_engagement_lineaire : MOTION_INSTRUCTION;
   Degagement_en_pos_demande : BOOL;
   MAS_degagement_maitreVnul : MOTION_INSTRUCTION;
   Engagement_came_VNul : BOOL;
   MCCP_First_Vnul : MOTION_INSTRUCTION;
   MCSV_Slave_Value : REAL;
   MCSV_Slope_Value : REAL;
   MCSV_SlopeD_Value : REAL;
   MCSV : MOTION_INSTRUCTION;
   MAM_engagement_lineaire_vnul : MOTION_INSTRUCTION;
   MAM_engagement_rotatifvnul : MOTION_INSTRUCTION;
   Val_MAitre : REAL;
   MAPC_First_Vnul : MOTION_INSTRUCTION;
   Front_vnul : BOOL;
   Val_Phase_Modulo2 : REAL;
   MCCP_1_vnul : MOTION_INSTRUCTION;
   Came_Prof_1_vnul : CAM_PROFILE[100];
   MAPC_1_vnul : MOTION_INSTRUCTION;
   MCCP_2_vnul : MOTION_INSTRUCTION;
   Came_Prof_2_vnul : CAM_PROFILE[100];
   MAPC_2_vnul : MOTION_INSTRUCTION;
   TEMP_5 : BOOL;
   Top_Calage5 : BOOL;
   TEMP_6 : BOOL;
   Top_Calage6 : BOOL;
   Erreur_3 : BOOL;
   Erreur_4 : BOOL;
   Front200 : BOOL;
   Cam_Pending : BOOL;
   Tempo_degagement : TIMER;
   decalage_Vnul_Dem : REAL;
   decalage_Vnul_Dem_modulo : REAL;
   front_degagement : BOOL; {access None}
   modulo_div2 : REAL; {access None}
   MCCP_First_Once : MOTION_INSTRUCTION; {access None}
   Came_Prof_First_Once : CAM_PROFILE[100]; {access None}
   MAPC_First_Once : MOTION_INSTRUCTION; {access None}
   Front_once : BOOL; {access None}
   Val_Engagement_plus_min : REAL; {access None}
   Synchro_0 : BOOL; {access None}
   Synchro_1 : BOOL; {access None}
   Val_Engagement_moins_min : REAL; {access None}
   TOF_MAPC_Actif : TIMER; {access None}
   Front_MAPC2 : BOOL; {access None}
   Front_MAPC1 : BOOL; {access None}
   Synchro_vnul_0 : BOOL; {access None}
   Synchro_vnul_1 : BOOL; {access None}
END_VAR

ROUTINE Logic   (* ladder *)
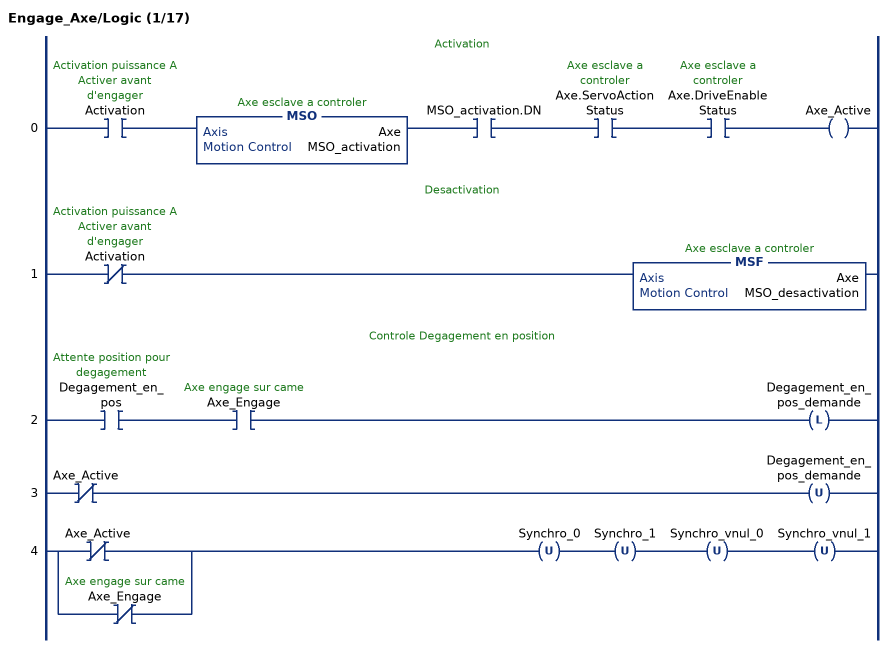
   // Activation
   0: XIC(Activation)MSO(Axe,MSO_activation)XIC(MSO_activation.DN)XIC(Axe.ServoActionStatus)XIC(Axe.DriveEnableStatus)OTE(Axe_Active);
   // Desactivation
   1: XIO(Activation)MSF(Axe,MSO_desactivation);
   // Controle Degagement en position
   2: XIC(Degagement_en_pos)XIC(Axe_Engage)OTL(Degagement_en_pos_demande);
   3: XIO(Axe_Active)OTU(Degagement_en_pos_demande);
   4: [XIO(Axe_Active) ,XIO(Axe_Engage) ]OTU(Synchro_0)OTU(Synchro_1)OTU(Synchro_vnul_0)OTU(Synchro_vnul_1);
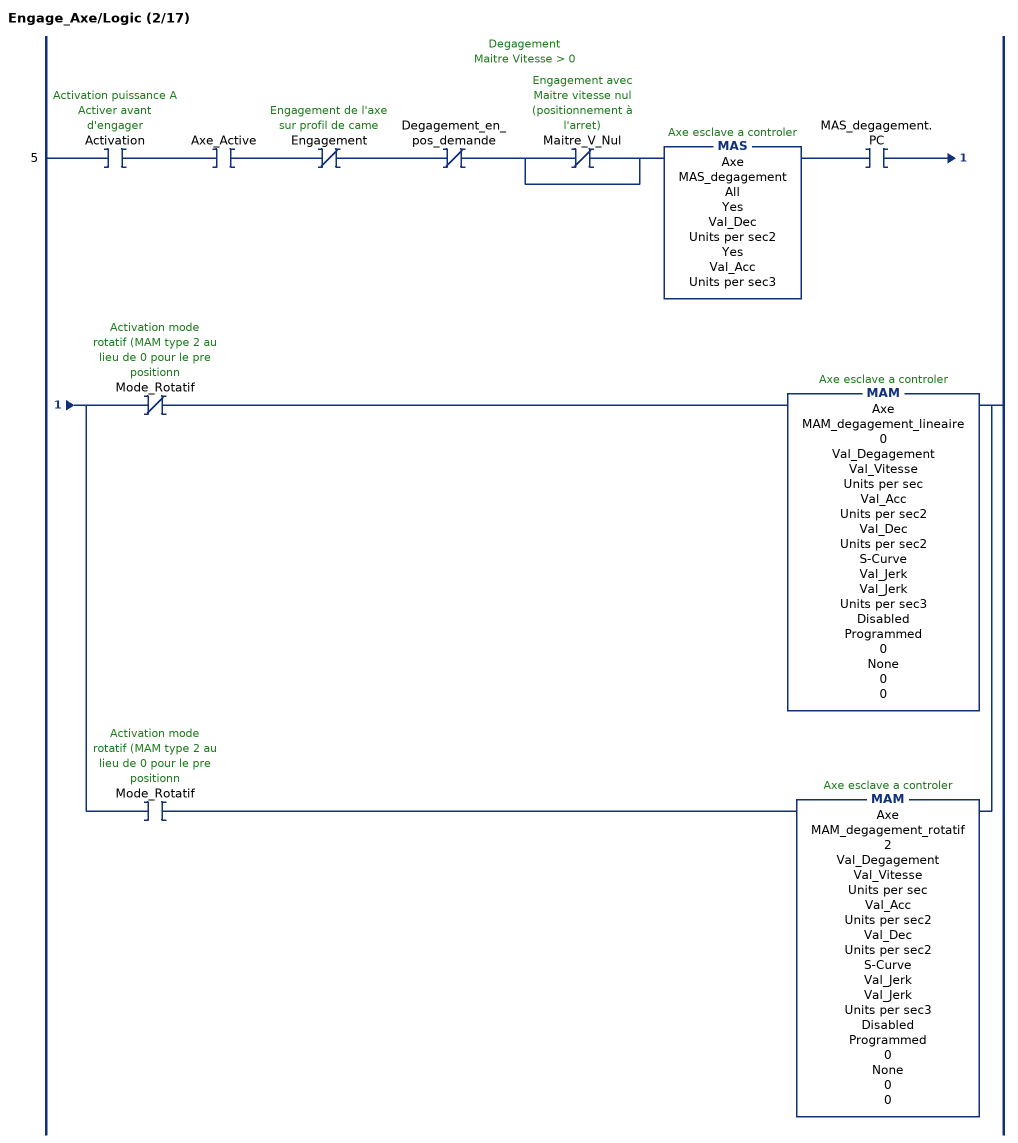
   // Degagement
   // Maitre Vitesse > 0
   5: XIC(Activation)XIC(Axe_Active)XIO(Engagement)XIO(Degagement_en_pos_demande)[XIO(Maitre_V_Nul) ,]MAS(Axe,MAS_degagement,All,Yes,Val_Dec,Units per sec2,Yes,Val_Acc,Units per sec3)XIC(MAS_degagement.PC)[XIO(Mode_Rotatif) MAM(Axe,MAM_degagement_lineaire,0,Val_Degagement,Val_Vitesse,Units per sec,Val_Acc,Units per sec2,Val_Dec,Units per sec2,S-Curve,Val_Jerk,Val_Jerk,Units per sec3,Disabled,Programmed,0,None,0,0) ,XIC(Mode_Rotatif) MAM(Axe,MAM_degagement_rotatif,2,Val_Degagement,Val_Vitesse,Units per sec,Val_Acc,Units per sec2,Val_Dec,Units per sec2,S-Curve,Val_Jerk,Val_Jerk,Units per sec3,Disabled,Programmed,0,None,0,0) ];
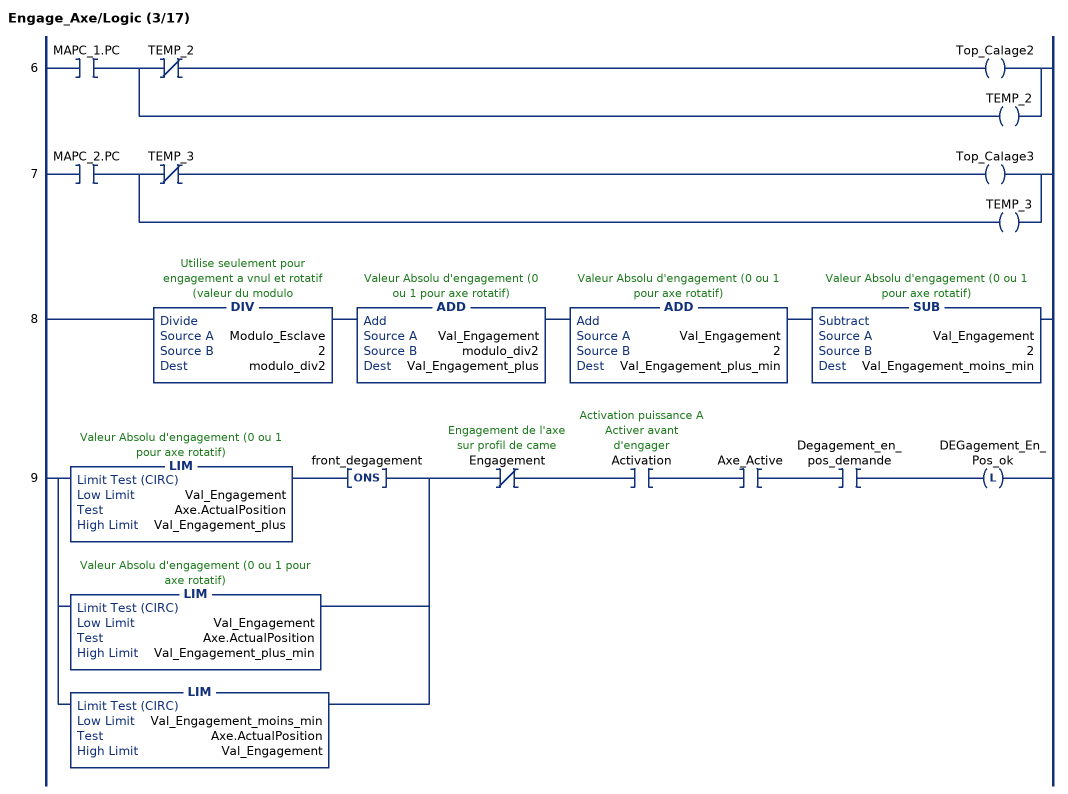
   6: XIC(MAPC_1.PC)[XIO(TEMP_2) OTE(Top_Calage2) ,OTE(TEMP_2) ];
   7: XIC(MAPC_2.PC)[XIO(TEMP_3) OTE(Top_Calage3) ,OTE(TEMP_3) ];
   8: DIV(Modulo_Esclave,2,modulo_div2)ADD(Val_Engagement,modulo_div2,Val_Engagement_plus)ADD(Val_Engagement,2,Val_Engagement_plus_min)SUB(Val_Engagement,2,Val_Engagement_moins_min);
   9: [LIM(Val_Engagement,Axe.ActualPosition,Val_Engagement_plus) ONS(front_degagement) ,LIM(Val_Engagement,Axe.ActualPosition,Val_Engagement_plus_min) ,LIM(Val_Engagement_moins_min,Axe.ActualPosition,Val_Engagement) ]XIO(Engagement)XIC(Activation)XIC(Axe_Active)XIC(Degagement_en_pos_demande)OTL(DEGagement_En_Pos_ok);
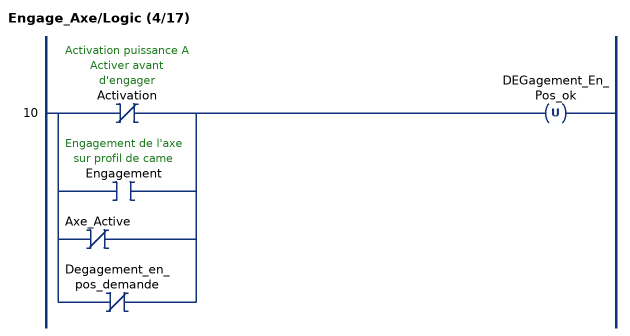
   10: [XIO(Activation) ,XIC(Engagement) ,XIO(Axe_Active) ,XIO(Degagement_en_pos_demande) ]OTU(DEGagement_En_Pos_ok);
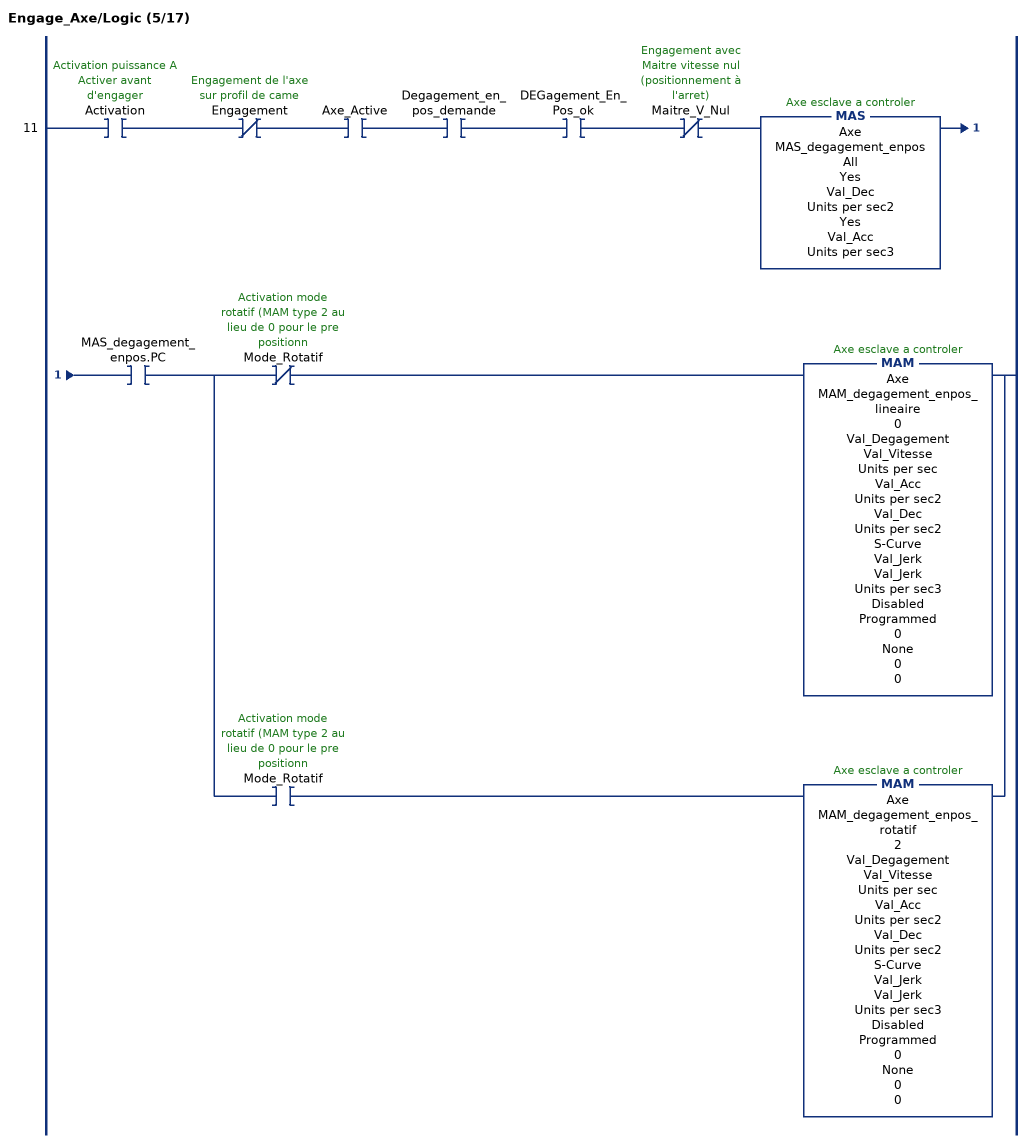
   11: XIC(Activation)XIO(Engagement)XIC(Axe_Active)XIC(Degagement_en_pos_demande)XIC(DEGagement_En_Pos_ok)XIO(Maitre_V_Nul)MAS(Axe,MAS_degagement_enpos,All,Yes,Val_Dec,Units per sec2,Yes,Val_Acc,Units per sec3)XIC(MAS_degagement_enpos.PC)[XIO(Mode_Rotatif) MAM(Axe,MAM_degagement_enpos_lineaire,0,Val_Degagement,Val_Vitesse,Units per sec,Val_Acc,Units per sec2,Val_Dec,Units per sec2,S-Curve,Val_Jerk,Val_Jerk,Units per sec3,Disabled,Programmed,0,None,0,0) ,XIC(Mode_Rotatif) MAM(Axe,MAM_degagement_enpos_rotatif,2,Val_Degagement,Val_Vitesse,Units per sec,Val_Acc,Units per sec2,Val_Dec,Units per sec2,S-Curve,Val_Jerk,Val_Jerk,Units per sec3,Disabled,Programmed,0,None,0,0) ];
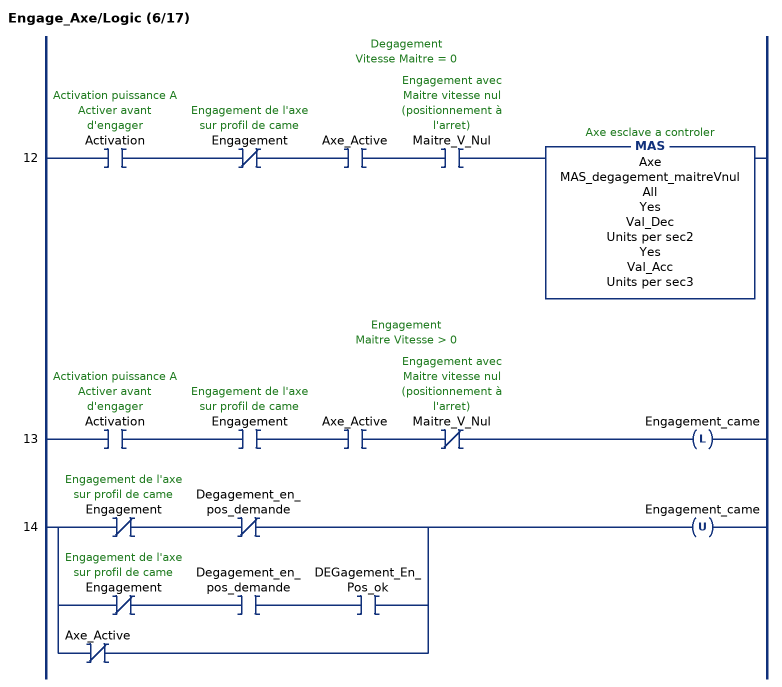
   // Degagement
   // Vitesse Maitre = 0
   12: XIC(Activation)XIO(Engagement)XIC(Axe_Active)XIC(Maitre_V_Nul)MAS(Axe,MAS_degagement_maitreVnul,All,Yes,Val_Dec,Units per sec2,Yes,Val_Acc,Units per sec3);
   // Engagement
   // Maitre Vitesse > 0
   13: XIC(Activation)XIC(Engagement)XIC(Axe_Active)XIO(Maitre_V_Nul)OTL(Engagement_came);
   14: [XIO(Engagement) XIO(Degagement_en_pos_demande) ,XIO(Engagement) XIC(Degagement_en_pos_demande) XIC(DEGagement_En_Pos_ok) ,XIO(Axe_Active) ]OTU(Engagement_came);
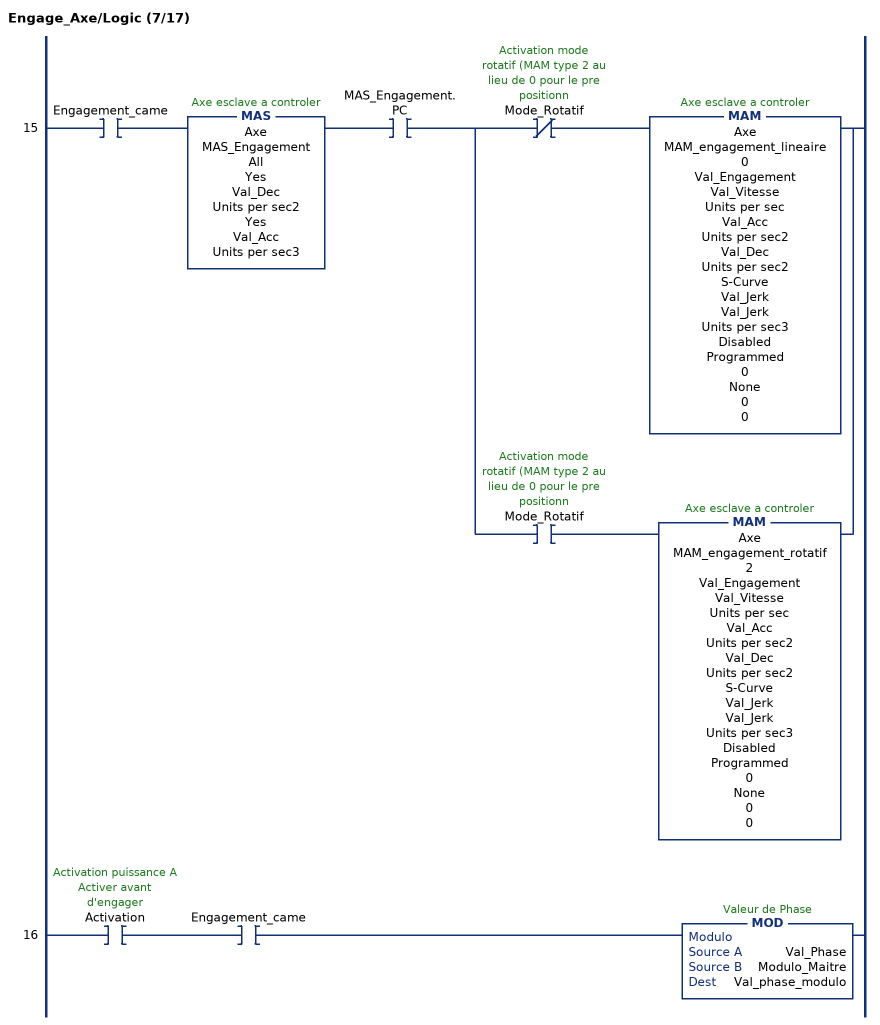
   15: XIC(Engagement_came)MAS(Axe,MAS_Engagement,All,Yes,Val_Dec,Units per sec2,Yes,Val_Acc,Units per sec3)XIC(MAS_Engagement.PC)[XIO(Mode_Rotatif) MAM(Axe,MAM_engagement_lineaire,0,Val_Engagement,Val_Vitesse,Units per sec,Val_Acc,Units per sec2,Val_Dec,Units per sec2,S-Curve,Val_Jerk,Val_Jerk,Units per sec3,Disabled,Programmed,0,None,0,0) ,XIC(Mode_Rotatif) MAM(Axe,MAM_engagement_rotatif,2,Val_Engagement,Val_Vitesse,Units per sec,Val_Acc,Units per sec2,Val_Dec,Units per sec2,S-Curve,Val_Jerk,Val_Jerk,Units per sec3,Disabled,Programmed,0,None,0,0) ];
   16: XIC(Activation)XIC(Engagement_came)MOD(Val_Phase,Modulo_Maitre,Val_phase_modulo);
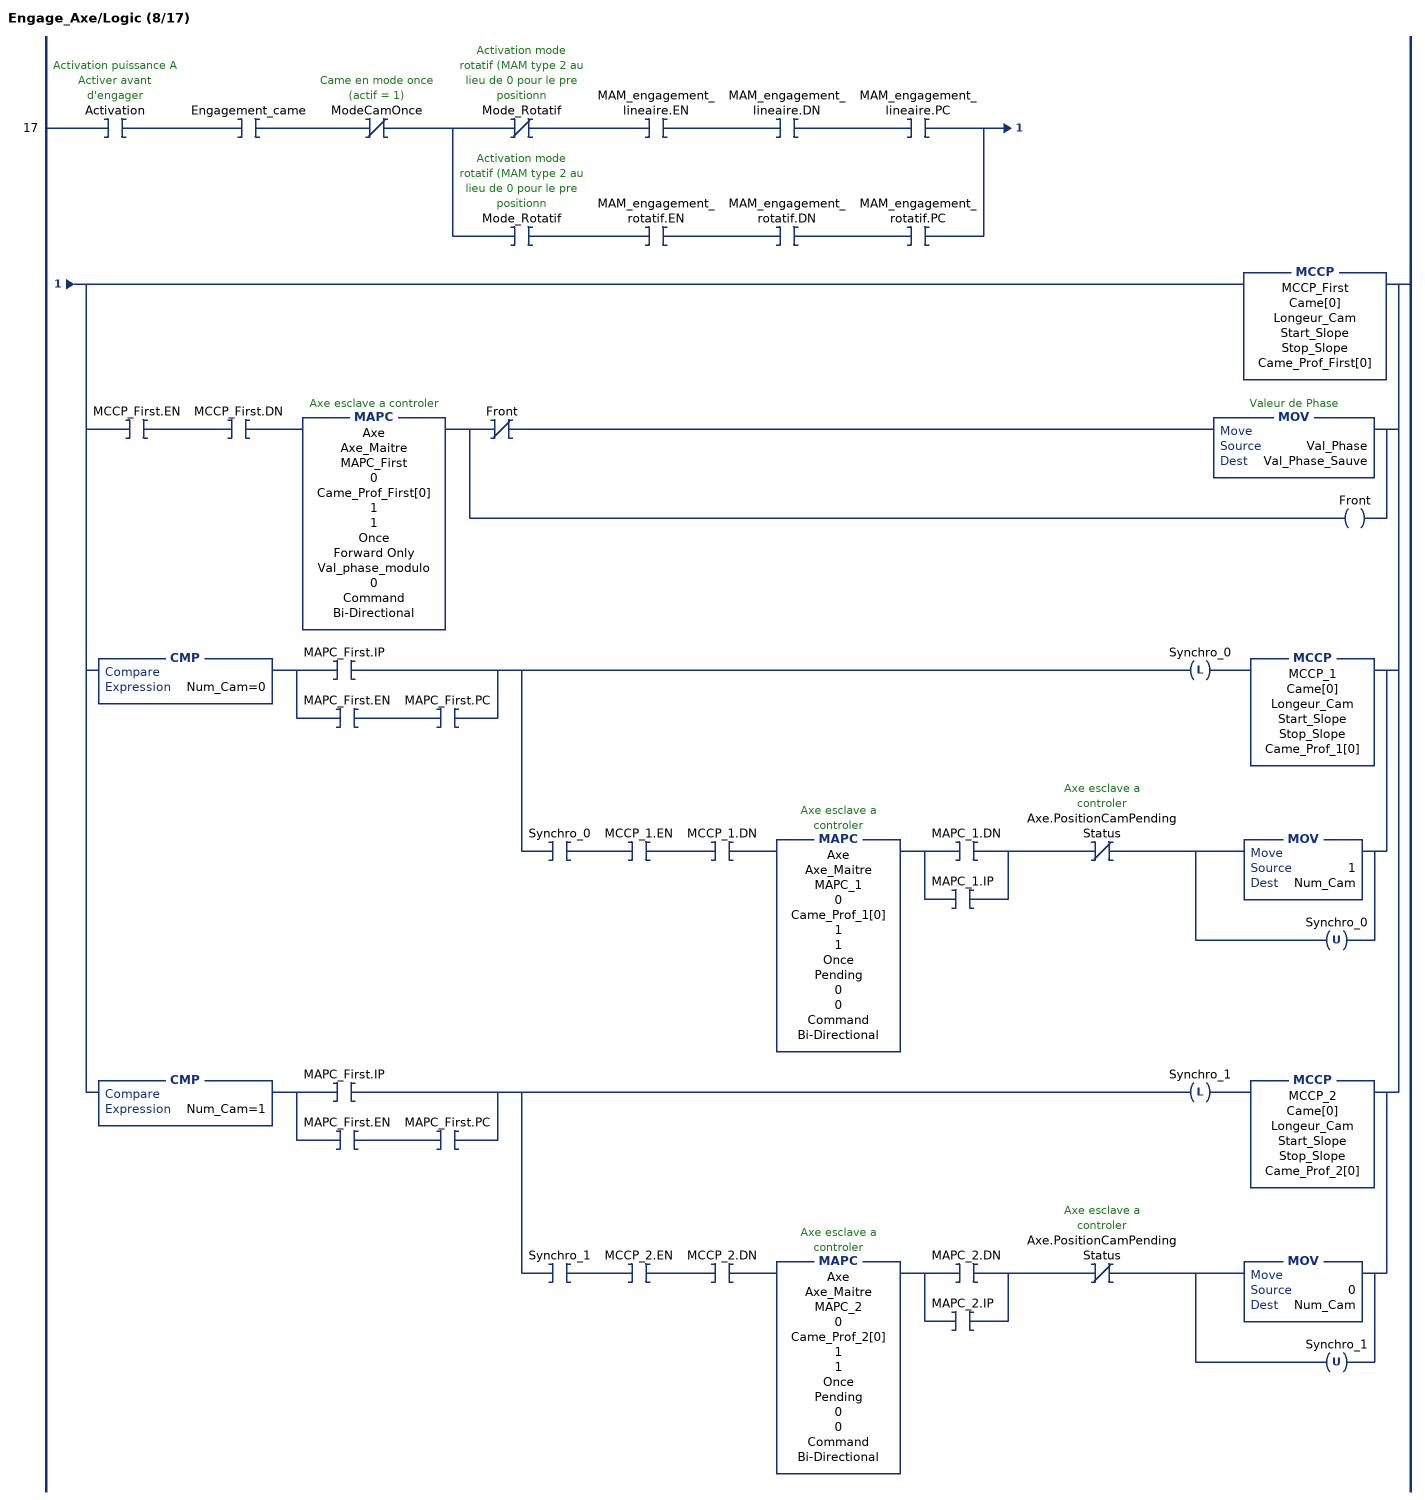
   17: XIC(Activation)XIC(Engagement_came)XIO(ModeCamOnce)[XIO(Mode_Rotatif) XIC(MAM_engagement_lineaire.EN) XIC(MAM_engagement_lineaire.DN) XIC(MAM_engagement_lineaire.PC) ,XIC(Mode_Rotatif) XIC(MAM_engagement_rotatif.EN) XIC(MAM_engagement_rotatif.DN) XIC(MAM_engagement_rotatif.PC) ][MCCP(MCCP_First,Came[0],Longeur_Cam,Start_Slope,Stop_Slope,Came_Prof_First[0]) ,[XIC(MCCP_First.EN) XIC(MCCP_First.DN) MAPC(Axe,Axe_Maitre,MAPC_First,0,Came_Prof_First[0],1,1,Once,Forward Only,Val_phase_modulo,0,Command,Bi-Directional) [XIO(Front) MOV(Val_Phase,Val_Phase_Sauve) ,OTE(Front) ] ,CMP(Num_Cam=0) [XIC(MAPC_First.IP) ,XIC(MAPC_First.EN) XIC(MAPC_First.PC) ] [OTL(Synchro_0) MCCP(MCCP_1,Came[0],Longeur_Cam,Start_Slope,Stop_Slope,Came_Prof_1[0]) ,XIC(Synchro_0) XIC(MCCP_1.EN) XIC(MCCP_1.DN) MAPC(Axe,Axe_Maitre,MAPC_1,0,Came_Prof_1[0],1,1,Once,Pending,0,0,Command,Bi-Directional) [XIC(MAPC_1.DN) ,XIC(MAPC_1.IP) ] XIO(Axe.PositionCamPendingStatus) [MOV(1,Num_Cam) ,OTU(Synchro_0) ] ] ,CMP(Num_Cam=1) [XIC(MAPC_First.IP) ,XIC(MAPC_First.EN) XIC(MAPC_First.PC) ] [OTL(Synchro_1) MCCP(MCCP_2,Came[0],Longeur_Cam,Start_Slope,Stop_Slope,Came_Prof_2[0]) ,XIC(Synchro_1) XIC(MCCP_2.EN) XIC(MCCP_2.DN) MAPC(Axe,Axe_Maitre,MAPC_2,0,Came_Prof_2[0],1,1,Once,Pending,0,0,Command,Bi-Directional) [XIC(MAPC_2.DN) ,XIC(MAPC_2.IP) ] XIO(Axe.PositionCamPendingStatus) [MOV(0,Num_Cam) ,OTU(Synchro_1) ] ] ] ];
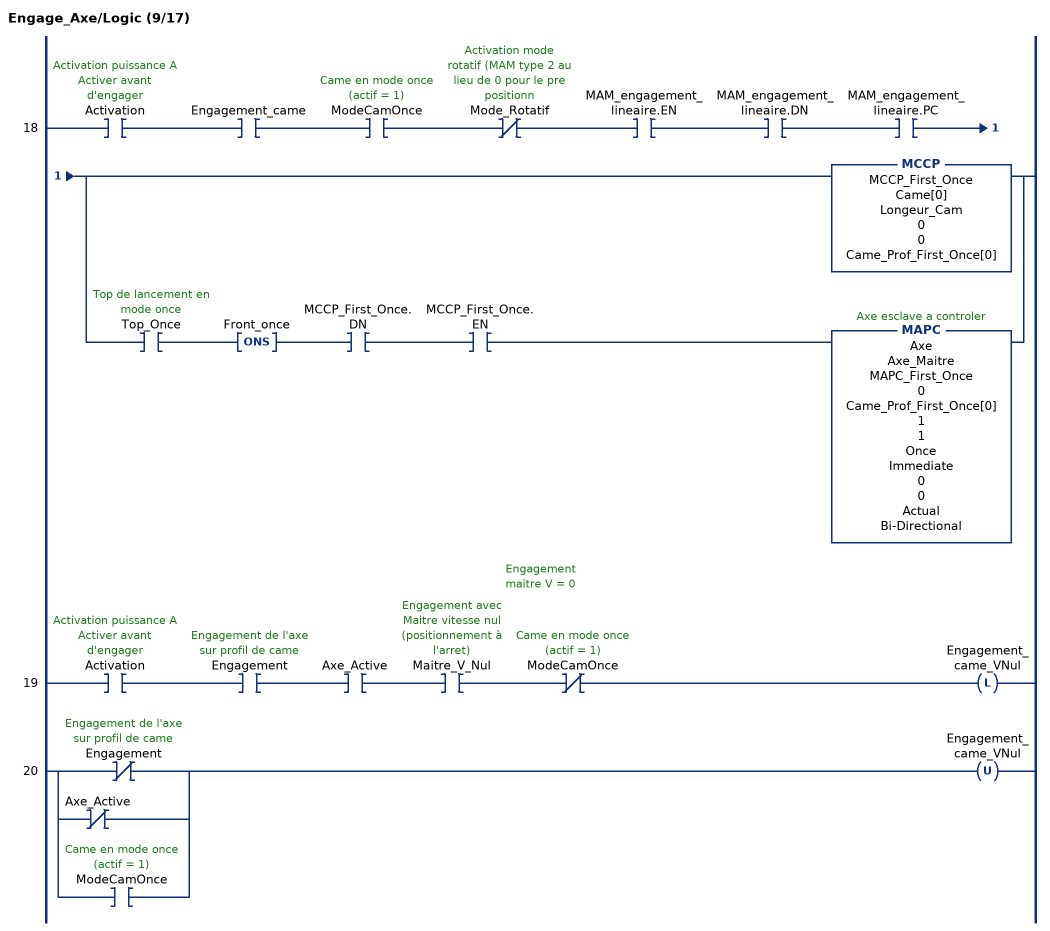
   18: XIC(Activation)XIC(Engagement_came)XIC(ModeCamOnce)XIO(Mode_Rotatif)XIC(MAM_engagement_lineaire.EN)XIC(MAM_engagement_lineaire.DN)XIC(MAM_engagement_lineaire.PC)[MCCP(MCCP_First_Once,Came[0],Longeur_Cam,0,0,Came_Prof_First_Once[0]) ,XIC(Top_Once) ONS(Front_once) XIC(MCCP_First_Once.DN) XIC(MCCP_First_Once.EN) MAPC(Axe,Axe_Maitre,MAPC_First_Once,0,Came_Prof_First_Once[0],1,1,Once,Immediate,0,0,Actual,Bi-Directional) ];
   // Engagement
   // maitre V = 0
   19: XIC(Activation)XIC(Engagement)XIC(Axe_Active)XIC(Maitre_V_Nul)XIO(ModeCamOnce)OTL(Engagement_came_VNul);
   20: [XIO(Engagement) ,XIO(Axe_Active) ,XIC(ModeCamOnce) ]OTU(Engagement_came_VNul);
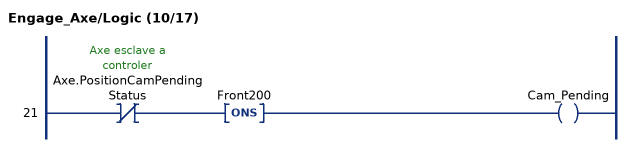
   21: XIO(Axe.PositionCamPendingStatus)ONS(Front200)OTE(Cam_Pending);
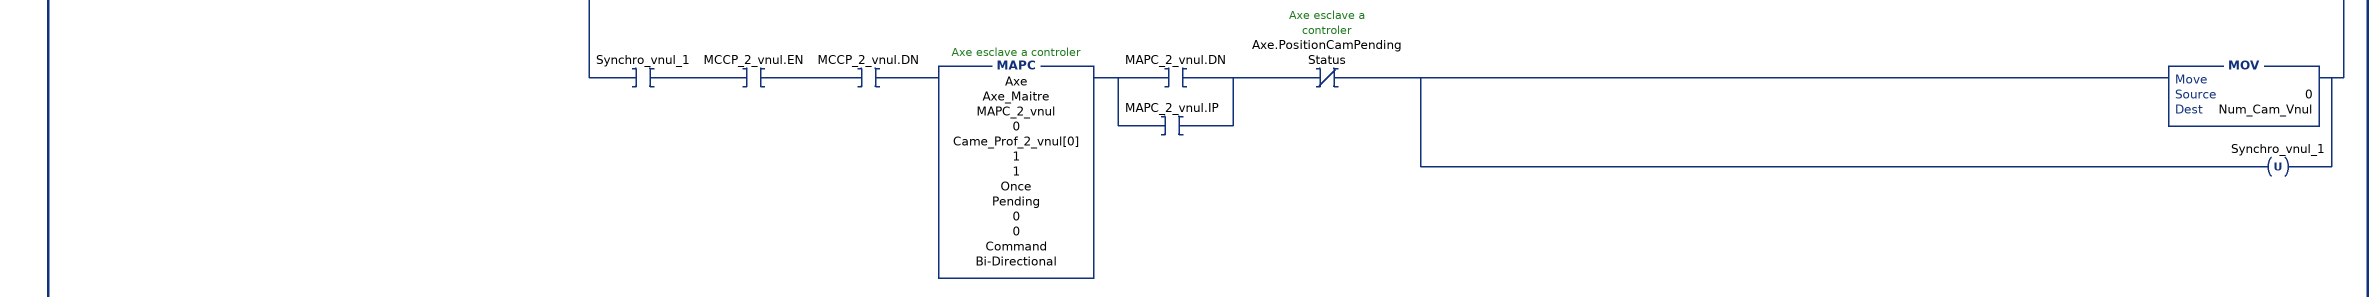
   22: XIC(Engagement_came_VNul)[MCCP(MCCP_First_Vnul,Came[0],Longeur_Cam,0,0,Came_Prof_First[0]) ,XIC(MCCP_First_Vnul.EN) XIC(MCCP_First_Vnul.DN) MOD(Val_Phase,Modulo_Maitre,Val_Phase_Modulo2) SUB(Axe_Maitre.CommandPosition,Val_Phase_Modulo2,Val_MAitre) ADD(Val_MAitre,Modulo_Maitre,Val_MAitre) MOD(Val_MAitre,Modulo_Maitre,Val_MAitre) MCSV(MCSV,Came_Prof_First[0],Val_MAitre,MCSV_Slave_Value,MCSV_Slope_Value,MCSV_SlopeD_Value) ADD(MCSV_Slave_Value,Val_Engagement,decalage_Vnul_Dem) MOD(decalage_Vnul_Dem,Modulo_Esclave,decalage_Vnul_Dem_modulo) XIC(MCSV.DN) [XIO(Mode_Rotatif) MAM(Axe,MAM_engagement_lineaire_vnul,0,decalage_Vnul_Dem,Val_Vitesse,Units per sec,Val_Acc,Units per sec2,Val_Dec,Units per sec2,S-Curve,Val_Jerk,Val_Jerk,Units per sec3,Disabled,Programmed,0,None,0,0) ,XIC(Mode_Rotatif) MAM(Axe,MAM_engagement_rotatifvnul,2,decalage_Vnul_Dem_modulo,Val_Vitesse,Units per sec,Val_Acc,Units per sec2,Val_Dec,Units per sec2,S-Curve,Val_Jerk,Val_Jerk,Units per sec3,Disabled,Programmed,0,None,0,0) ] ,XIC(MCCP_First_Vnul.EN) XIC(MCCP_First_Vnul.DN) MAPC(Axe,Axe_Maitre,MAPC_First_Vnul,0,Came_Prof_First[0],1,1,Once,Immediate,0,Val_MAitre,Command,Bi-Directional) [XIO(Front_vnul) MOV(Val_Phase,Val_Phase_Sauve) ,OTE(Front_vnul) ] ,CMP(Num_Cam_Vnul=0) [XIC(MAPC_First_Vnul.IP) ,XIC(MAPC_First_Vnul.EN) XIC(MAPC_First_Vnul.PC) ] [OTL(Synchro_vnul_0) MCCP(MCCP_1_vnul,Came[0],Longeur_Cam,0,0,Came_Prof_1_vnul[0]) ,XIC(Synchro_vnul_0) XIC(MCCP_1_vnul.EN) XIC(MCCP_1_vnul.DN) MAPC(Axe,Axe_Maitre,MAPC_1_vnul,0,Came_Prof_1_vnul[0],1,1,Once,Pending,0,0,Command,Bi-Directional) [XIC(MAPC_1_vnul.DN) ,XIC(MAPC_1_vnul.IP) ] XIO(Axe.PositionCamPendingStatus) [MOV(1,Num_Cam_Vnul) ,OTU(Synchro_vnul_0) ] ] ,CMP(Num_Cam_Vnul=1) [XIC(MAPC_First_Vnul.IP) ,XIC(MAPC_First_Vnul.EN) XIC(MAPC_First_Vnul.PC) ] [OTL(Synchro_vnul_1) MCCP(MCCP_2_vnul,Came[0],Longeur_Cam,0,0,Came_Prof_2_vnul[0]) ,XIC(Synchro_vnul_1) XIC(MCCP_2_vnul.EN) XIC(MCCP_2_vnul.DN) MAPC(Axe,Axe_Maitre,MAPC_2_vnul,0,Came_Prof_2_vnul[0],1,1,Once,Pending,0,0,Command,Bi-Directional) [XIC(MAPC_2_vnul.DN) ,XIC(MAPC_2_vnul.IP) ] XIO(Axe.PositionCamPendingStatus) [MOV(0,Num_Cam_Vnul) ,OTU(Synchro_vnul_1) ] ] ];
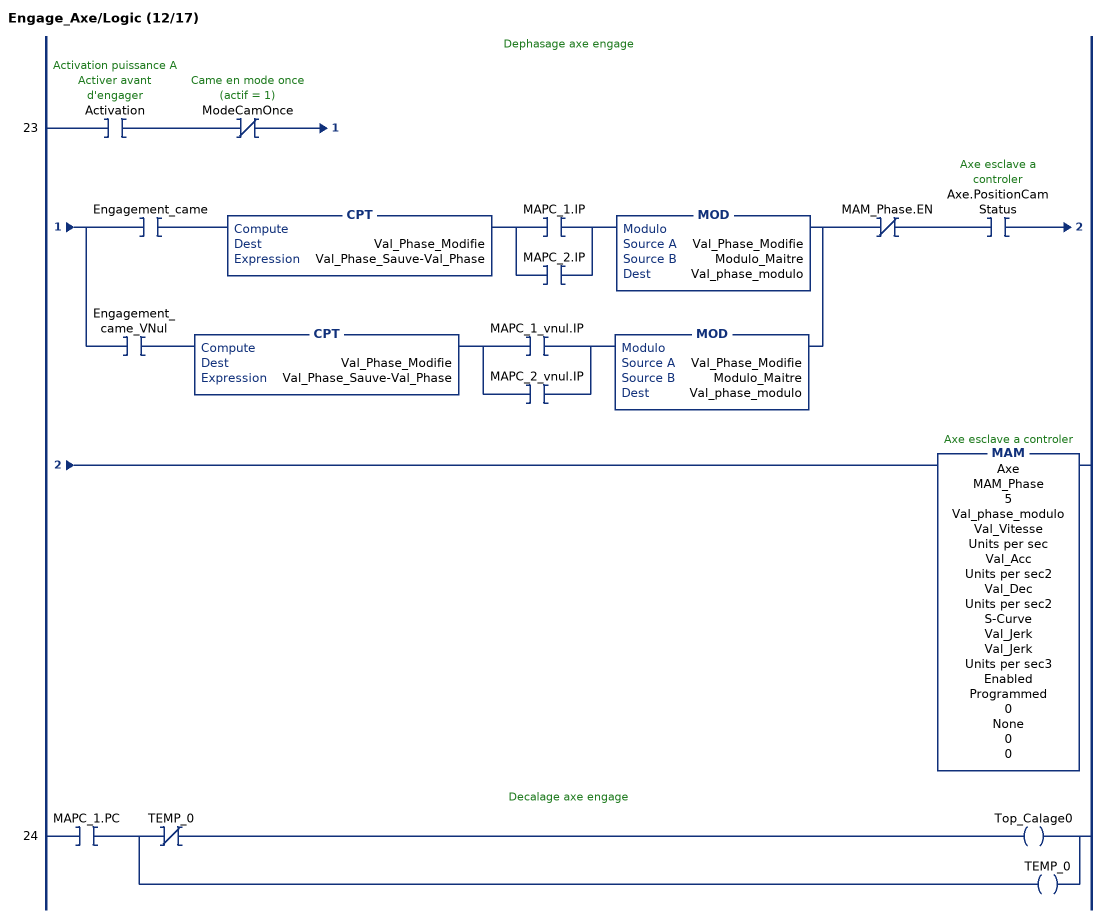
   // Dephasage axe engage
   23: XIC(Activation)XIO(ModeCamOnce)[XIC(Engagement_came) CPT(Val_Phase_Modifie,Val_Phase_Sauve-Val_Phase) [XIC(MAPC_1.IP) ,XIC(MAPC_2.IP) ] MOD(Val_Phase_Modifie,Modulo_Maitre,Val_phase_modulo) ,XIC(Engagement_came_VNul) CPT(Val_Phase_Modifie,Val_Phase_Sauve-Val_Phase) [XIC(MAPC_1_vnul.IP) ,XIC(MAPC_2_vnul.IP) ] MOD(Val_Phase_Modifie,Modulo_Maitre,Val_phase_modulo) ]XIO(MAM_Phase.EN)XIC(Axe.PositionCamStatus)MAM(Axe,MAM_Phase,5,Val_phase_modulo,Val_Vitesse,Units per sec,Val_Acc,Units per sec2,Val_Dec,Units per sec2,S-Curve,Val_Jerk,Val_Jerk,Units per sec3,Enabled,Programmed,0,None,0,0);
   // Decalage axe engage
   24: XIC(MAPC_1.PC)[XIO(TEMP_0) OTE(Top_Calage0) ,OTE(TEMP_0) ];
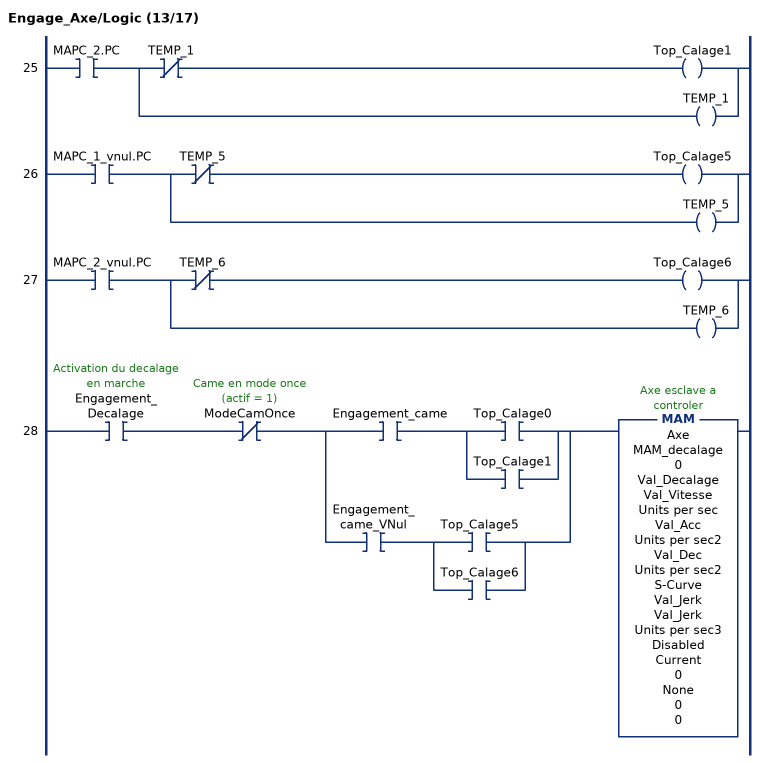
   25: XIC(MAPC_2.PC)[XIO(TEMP_1) OTE(Top_Calage1) ,OTE(TEMP_1) ];
   26: XIC(MAPC_1_vnul.PC)[XIO(TEMP_5) OTE(Top_Calage5) ,OTE(TEMP_5) ];
   27: XIC(MAPC_2_vnul.PC)[XIO(TEMP_6) OTE(Top_Calage6) ,OTE(TEMP_6) ];
   28: XIC(Engagement_Decalage)XIO(ModeCamOnce)[XIC(Engagement_came) [XIC(Top_Calage0) ,XIC(Top_Calage1) ] ,XIC(Engagement_came_VNul) [XIC(Top_Calage5) ,XIC(Top_Calage6) ] ]MAM(Axe,MAM_decalage,0,Val_Decalage,Val_Vitesse,Units per sec,Val_Acc,Units per sec2,Val_Dec,Units per sec2,S-Curve,Val_Jerk,Val_Jerk,Units per sec3,Disabled,Current,0,None,0,0);
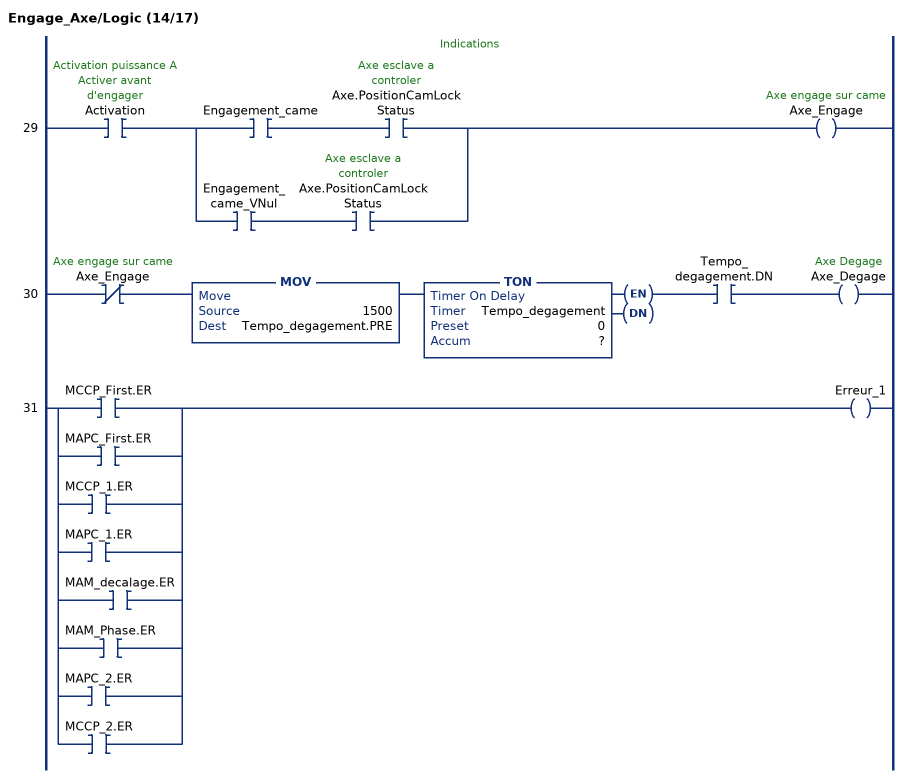
   // Indications
   29: XIC(Activation)[XIC(Engagement_came) XIC(Axe.PositionCamLockStatus) ,XIC(Engagement_came_VNul) XIC(Axe.PositionCamLockStatus) ]OTE(Axe_Engage);
   30: XIO(Axe_Engage)MOV(1500,Tempo_degagement.PRE)TON(Tempo_degagement,?,?)XIC(Tempo_degagement.DN)OTE(Axe_Degage);
   31: [XIC(MCCP_First.ER) ,XIC(MAPC_First.ER) ,XIC(MCCP_1.ER) ,XIC(MAPC_1.ER) ,XIC(MAM_decalage.ER) ,XIC(MAM_Phase.ER) ,XIC(MAPC_2.ER) ,XIC(MCCP_2.ER) ]OTE(Erreur_1);
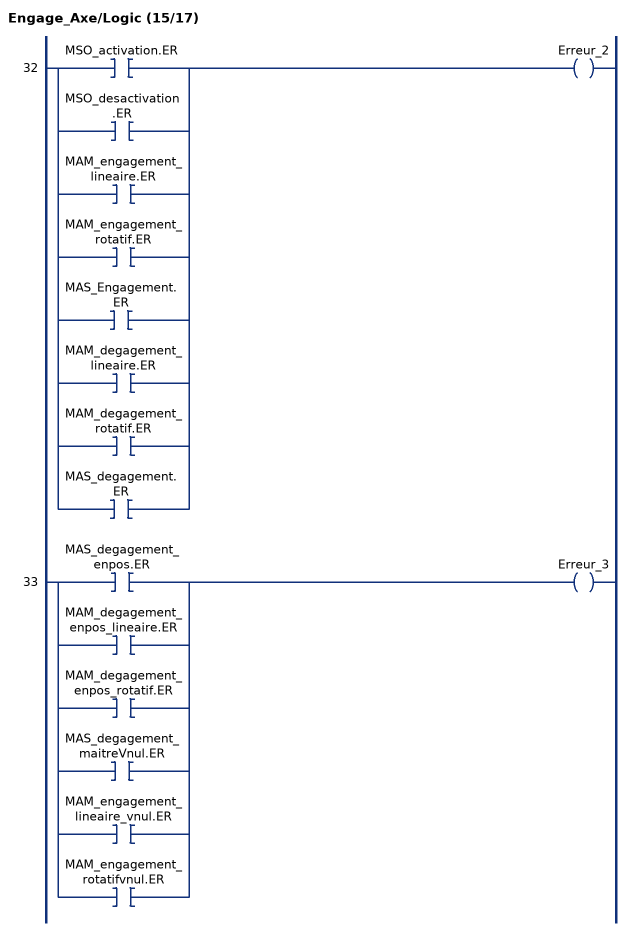
   32: [XIC(MSO_activation.ER) ,XIC(MSO_desactivation.ER) ,[XIC(MAM_engagement_lineaire.ER) ,XIC(MAM_engagement_rotatif.ER) ] ,XIC(MAS_Engagement.ER) ,[XIC(MAM_degagement_lineaire.ER) ,XIC(MAM_degagement_rotatif.ER) ] ,XIC(MAS_degagement.ER) ]OTE(Erreur_2);
   33: [XIC(MAS_degagement_enpos.ER) ,[XIC(MAM_degagement_enpos_lineaire.ER) ,[XIC(MAM_degagement_enpos_rotatif.ER) ,[XIC(MAS_degagement_maitreVnul.ER) ,[XIC(MAM_engagement_lineaire_vnul.ER) ,XIC(MAM_engagement_rotatifvnul.ER) ] ] ] ] ]OTE(Erreur_3);
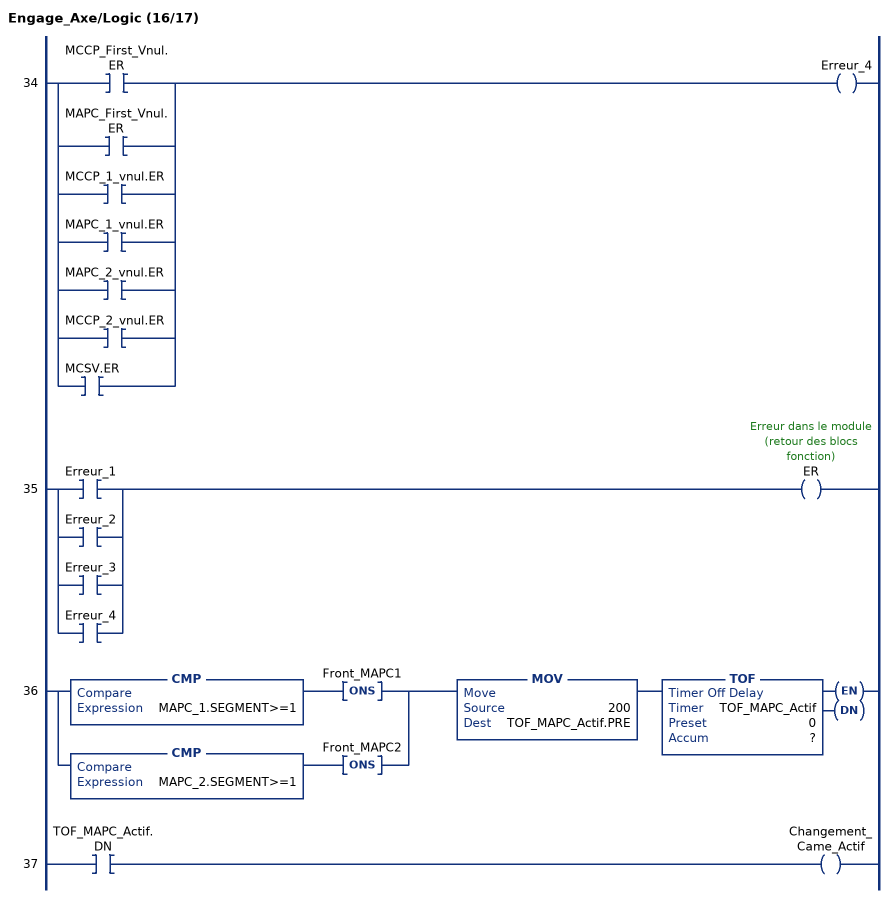
   34: [XIC(MCCP_First_Vnul.ER) ,XIC(MAPC_First_Vnul.ER) ,XIC(MCCP_1_vnul.ER) ,XIC(MAPC_1_vnul.ER) ,XIC(MAPC_2_vnul.ER) ,XIC(MCCP_2_vnul.ER) ,XIC(MCSV.ER) ]OTE(Erreur_4);
   35: [XIC(Erreur_1) ,XIC(Erreur_2) ,XIC(Erreur_3) ,XIC(Erreur_4) ]OTE(ER);
   36: [CMP(MAPC_1.SEGMENT>=1) ONS(Front_MAPC1) ,CMP(MAPC_2.SEGMENT>=1) ONS(Front_MAPC2) ]MOV(200,TOF_MAPC_Actif.PRE)TOF(TOF_MAPC_Actif,?,?);
   37: XIC(TOF_MAPC_Actif.DN)OTE(Changement_Came_Actif);
